SPLINE
SPL {X  -158.454, Y  +360.384, Z    +0.000, E1  +340.634, E3 -429443.801}
SPL {X  -159.737, Y  +373.507, Z    +0.000, E1  +349.689, E3 -429465.837}
SPL {X  -159.990, Y  +382.574, Z    +0.000, E1  +355.537, E3 -429472.525}
SPL {X  -159.990, Y  +389.909, Z    +0.000, E1  +360.662, E3 -429476.539}
SPL {X  -159.990, Y  +396.289, Z    +0.000, E1  +365.500, E3 -429480.319}
SPL {X  -159.990, Y  +407.941, Z    +0.000, E1  +374.126, E3 -429491.656}
SPL {X  -159.990, Y  +418.671, Z    +0.000, E1  +379.855, E3 -429511.072}
SPL {X  -159.990, Y  +429.878, Z    +0.000, E1  +383.330, E3 -429541.127}
SPL {X  -159.990, Y  +432.766, Z    +0.000, E1  +383.321, E3 -429555.350}
SPL {X  -159.990, Y  +434.794, Z    +0.000, E1  +383.304, E3 -429565.381}
SPL {X  -159.990, Y  +437.007, Z    +0.000, E1  +383.323, E3 -429576.234}
SPL {X  -159.990, Y  +439.778, Z    +0.000, E1  +383.323, E3 -429589.866}
SPL {X  -159.990, Y  +442.945, Z    +0.000, E1  +383.339, E3 -429605.430}
SPL {X  -159.990, Y  +446.037, Z    +0.000, E1  +383.324, E3 -429620.680}
SPL {X  -159.990, Y  +448.341, Z    +0.000, E1  +383.317, E3 -429631.998}
SPL {X  -159.990, Y  +450.345, Z    +0.000, E1  +383.316, E3 -429641.876}
SPL {X  -159.990, Y  +452.828, Z    +0.000, E1  +383.330, E3 -429654.075}
SPL {X  -159.990, Y  +456.338, Z    +0.000, E1  +383.359, E3 -429671.267}
SPL {X  -159.990, Y  +459.480, Z    +0.000, E1  +383.323, E3 -429686.809}
SPL {X  -159.990, Y  +461.803, Z    +0.000, E1  +383.322, E3 -429698.244}
SPL {X  -159.990, Y  +464.971, Z    +0.000, E1  +383.357, E3 -429713.750}
SPL {X  -159.990, Y  +467.934, Z    +0.000, E1  +383.321, E3 -429728.407}
SPL {X  -159.990, Y  +469.939, Z    +0.000, E1  +383.319, E3 -429738.269}
SPL {X  -159.990, Y  +472.144, Z    +0.000, E1  +383.327, E3 -429749.120}
SPL {X  -159.990, Y  +474.152, Z    +0.000, E1  +383.309, E3 -429759.072}
SPL {X  -159.990, Y  +475.762, Z    +0.000, E1  +383.308, E3 -429767.001}
SPL {X  -159.990, Y  +478.041, Z    +0.000, E1  +383.328, E3 -429778.177}
SPL {X  -159.990, Y  +480.905, Z    +0.000, E1  +383.327, E3 -429792.273}
SPL {X  -159.990, Y  +484.251, Z    +0.000, E1  +383.352, E3 -429808.688}
SPL {X  -159.990, Y  +488.031, Z    +0.000, E1  +383.345, E3 -429827.321}
SPL {X  -159.990, Y  +491.121, Z    +0.000, E1  +383.323, E3 -429842.567}
SPL {X  -159.990, Y  +493.610, Z    +0.000, E1  +383.323, E3 -429854.820}
SPL {X  -159.990, Y  +496.863, Z    +0.000, E1  +383.350, E3 -429870.780}
SPL {X  -159.990, Y  +499.995, Z    +0.000, E1  +383.324, E3 -429886.241}
SPL {X  -159.990, Y  +502.341, Z    +0.000, E1  +383.320, E3 -429897.800}
SPL {X  -159.990, Y  +505.377, Z    +0.000, E1  +383.346, E3 -429912.691}
SPL {X  -159.990, Y  +508.024, Z    +0.000, E1  +383.315, E3 -429925.773}
SPL {X  -159.990, Y  +510.344, Z    +0.000, E1  +383.327, E3 -429937.180}
SPL {X  -159.990, Y  +513.289, Z    +0.000, E1  +383.332, E3 -429951.670}
SPL {X  -159.990, Y  +516.195, Z    +0.000, E1  +383.325, E3 -429965.989}
SPL {X  -159.990, Y  +518.925, Z    +0.000, E1  +383.333, E3 -429979.352}
SPL {X  -159.990, Y  +521.408, Z    +0.000, E1  +383.329, E3 -429991.561}
SPL {X  -159.990, Y  +523.942, Z    +0.000, E1  +383.333, E3 -430004.054}
SPL {X  -159.990, Y  +526.221, Z    +0.000, E1  +383.314, E3 -430015.330}
SPL {X  -159.990, Y  +527.834, Z    +0.000, E1  +383.311, E3 -430023.280}
SPL {X  -159.990, Y  +529.993, Z    +0.000, E1  +383.329, E3 -430033.856}
SPL {X  -159.990, Y  +532.441, Z    +0.000, E1  +383.322, E3 -430045.907}
SPL {X  -159.990, Y  +534.618, Z    +0.000, E1  +383.322, E3 -430056.640}
SPL {X  -159.990, Y  +537.024, Z    +0.000, E1  +383.321, E3 -430068.502}
SPL {X  -159.990, Y  +539.129, Z    +0.000, E1  +383.310, E3 -430078.885}
SPL {X  -159.990, Y  +541.183, Z    +0.000, E1  +383.319, E3 -430088.982}
SPL {X  -159.990, Y  +543.647, Z    +0.000, E1  +383.325, E3 -430101.085}
SPL {X  -159.990, Y  +546.832, Z    +0.000, E1  +383.349, E3 -430116.708}
SPL {X  -159.990, Y  +549.756, Z    +0.000, E1  +383.320, E3 -430131.149}
SPL {X  -159.990, Y  +551.655, Z    +0.000, E1  +383.320, E3 -430140.499}
SPL {X  -159.990, Y  +553.711, Z    +0.000, E1  +383.317, E3 -430150.621}
SPL {X  -159.990, Y  +555.637, Z    +0.000, E1  +383.323, E3 -430160.090}
SPL {X  -159.990, Y  +558.758, Z    +0.000, E1  +383.351, E3 -430175.400}
SPL {X  -159.990, Y  +561.830, Z    +0.000, E1  +383.325, E3 -430190.573}
SPL {X  -159.990, Y  +564.273, Z    +0.000, E1  +383.325, E3 -430202.597}
SPL {X  -159.990, Y  +567.351, Z    +0.000, E1  +383.348, E3 -430217.693}
SPL {X  -159.990, Y  +570.314, Z    +0.000, E1  +383.326, E3 -430232.325}
SPL {X  -159.990, Y  +572.504, Z    +0.000, E1  +383.321, E3 -430243.110}
SPL {X  -159.990, Y  +575.653, Z    +0.000, E1  +383.355, E3 -430258.547}
SPL {X  -159.990, Y  +578.932, Z    +0.000, E1  +383.330, E3 -430274.730}
SPL {X  -159.990, Y  +581.497, Z    +0.000, E1  +383.329, E3 -430287.314}
SPL {X  -159.990, Y  +583.973, Z    +0.000, E1  +383.332, E3 -430299.499}
SPL {X  -159.990, Y  +586.877, Z    +0.000, E1  +383.349, E3 -430313.754}
SPL {X  -159.990, Y  +590.594, Z    +0.000, E1  +383.363, E3 -430332.004}
SPL {X  -159.990, Y  +593.847, Z    +0.000, E1  +383.340, E3 -430348.015}
SPL {X  -159.990, Y  +597.018, Z    +0.000, E1  +383.367, E3 -430363.546}
SPL {X  -159.990, Y  +599.887, Z    +0.000, E1  +383.341, E3 -430377.651}
SPL {X  -159.990, Y  +601.949, Z    +0.000, E1  +383.344, E3 -430387.777}
SPL {X  -159.990, Y  +605.106, Z    +0.000, E1  +383.383, E3 -430403.224}
SPL {X  -159.990, Y  +608.111, Z    +0.000, E1  +383.342, E3 -430418.075}
SPL {X  -159.990, Y  +610.073, Z    +0.000, E1  +383.343, E3 -430427.733}
SPL {X  -159.990, Y  +613.021, Z    +0.000, E1  +383.365, E3 -430442.203}
SPL {X  -159.990, Y  +615.657, Z    +0.000, E1  +383.331, E3 -430455.251}
SPL {X  -159.990, Y  +617.658, Z    +0.000, E1  +383.335, E3 -430465.093}
SPL {X  -159.990, Y  +620.788, Z    +0.000, E1  +383.368, E3 -430480.427}
SPL {X  -159.990, Y  +624.347, Z    +0.000, E1  +383.355, E3 -430497.947}
SPL {X  -159.990, Y  +627.144, Z    +0.000, E1  +383.340, E3 -430511.716}
SPL {X  -159.990, Y  +629.284, Z    +0.000, E1  +383.339, E3 -430522.224}
SPL {X  -159.990, Y  +631.206, Z    +0.000, E1  +383.337, E3 -430531.678}
SPL {X  -159.990, Y  +633.318, Z    +0.000, E1  +383.339, E3 -430542.082}
SPL {X  -159.990, Y  +635.650, Z    +0.000, E1  +383.339, E3 -430553.553}
SPL {X  -159.990, Y  +637.597, Z    +0.000, E1  +383.330, E3 -430563.176}
SPL {X  -159.990, Y  +640.369, Z    +0.000, E1  +383.354, E3 -430576.810}
SPL {X  -159.990, Y  +644.241, Z    +0.000, E1  +383.355, E3 -430595.922}
SPL {X  -159.990, Y  +648.287, Z    +0.000, E1  +383.349, E3 -430615.879}
SPL {X  -159.990, Y  +651.427, Z    +0.000, E1  +383.319, E3 -430631.374}
SPL {X  -159.990, Y  +653.536, Z    +0.000, E1  +383.313, E3 -430641.755}
SPL {X  -159.990, Y  +656.380, Z    +0.000, E1  +383.347, E3 -430655.691}
SPL {X  -159.990, Y  +659.180, Z    +0.000, E1  +383.314, E3 -430669.540}
SPL {X  -159.990, Y  +661.392, Z    +0.000, E1  +383.318, E3 -430680.433}
SPL {X  -159.990, Y  +663.662, Z    +0.000, E1  +383.322, E3 -430691.557}
SPL {X  -159.990, Y  +665.964, Z    +0.000, E1  +383.328, E3 -430702.848}
SPL {X  -159.990, Y  +668.989, Z    +0.000, E1  +383.359, E3 -430717.684}
SPL {X  -159.983, Y  +672.946, Z    +0.000, E1  +383.359, E3 -430737.165}
SPL {X  -159.924, Y  +676.110, Z    +0.000, E1  +383.320, E3 -430752.864}
SPL {X  -159.845, Y  +678.302, Z    +0.000, E1  +383.298, E3 -430763.766}
SPL {X  -159.760, Y  +680.081, Z    +0.000, E1  +383.288, E3 -430772.610}
SPL {X  -159.626, Y  +682.287, Z    +0.000, E1  +383.280, E3 -430783.581}
SPL {X  -159.462, Y  +684.486, Z    +0.000, E1  +383.258, E3 -430794.581}
SPL {X  -159.212, Y  +687.262, Z    +0.000, E1  +383.238, E3 -430808.485}
SPL {X  -158.971, Y  +689.529, Z    +0.000, E1  +383.181, E3 -430819.944}
SPL {X  -158.658, Y  +692.098, Z    +0.000, E1  +383.176, E3 -430832.851}
ENDSPLINE

SPLINE
SPL {X  -159.063, Y  +688.696, Z    +0.000, E1  +377.094, E3 -430875.070}
SPL {X  -159.987, Y  +672.488, Z    +0.000, E1  +365.638, E3 -430899.134}
SPL {X  -159.990, Y  +663.928, Z    +0.000, E1  +359.662, E3 -430904.929}
SPL {X  -159.990, Y  +658.009, Z    +0.000, E1  +355.226, E3 -430908.629}
SPL {X  -159.990, Y  +651.879, Z    +0.000, E1  +350.548, E3 -430913.691}
SPL {X  -159.990, Y  +637.832, Z    +0.000, E1  +341.694, E3 -430931.282}
SPL {X  -159.990, Y  +626.634, Z    +0.000, E1  +337.968, E3 -430962.136}
SPL {X  -159.990, Y  +624.622, Z    +0.000, E1  +337.980, E3 -430972.719}
SPL {X  -159.990, Y  +622.489, Z    +0.000, E1  +337.969, E3 -430983.886}
SPL {X  -159.990, Y  +619.955, Z    +0.000, E1  +337.968, E3 -430997.176}
SPL {X  -159.990, Y  +617.386, Z    +0.000, E1  +337.968, E3 -431010.650}
SPL {X  -159.990, Y  +614.863, Z    +0.000, E1  +337.969, E3 -431023.883}
SPL {X  -159.990, Y  +612.600, Z    +0.000, E1  +337.975, E3 -431035.767}
SPL {X  -159.990, Y  +610.646, Z    +0.000, E1  +337.979, E3 -431046.024}
SPL {X  -159.990, Y  +608.810, Z    +0.000, E1  +337.977, E3 -431055.657}
SPL {X  -159.990, Y  +605.804, Z    +0.000, E1  +337.936, E3 -431071.302}
SPL {X  -159.990, Y  +602.819, Z    +0.000, E1  +337.963, E3 -431086.974}
SPL {X  -159.990, Y  +600.642, Z    +0.000, E1  +337.968, E3 -431098.402}
SPL {X  -159.990, Y  +598.568, Z    +0.000, E1  +337.954, E3 -431109.194}
SPL {X  -159.990, Y  +595.493, Z    +0.000, E1  +337.930, E3 -431125.278}
SPL {X  -159.990, Y  +592.865, Z    +0.000, E1  +337.964, E3 -431139.106}
SPL {X  -159.990, Y  +590.803, Z    +0.000, E1  +337.954, E3 -431149.897}
SPL {X  -159.990, Y  +588.288, Z    +0.000, E1  +337.950, E3 -431163.061}
SPL {X  -159.990, Y  +586.040, Z    +0.000, E1  +337.954, E3 -431174.806}
SPL {X  -159.990, Y  +584.080, Z    +0.000, E1  +337.953, E3 -431185.066}
SPL {X  -159.990, Y  +581.924, Z    +0.000, E1  +337.949, E3 -431196.366}
SPL {X  -159.990, Y  +579.673, Z    +0.000, E1  +337.950, E3 -431208.165}
SPL {X  -159.990, Y  +576.961, Z    +0.000, E1  +337.936, E3 -431222.344}
SPL {X  -159.990, Y  +574.188, Z    +0.000, E1  +337.947, E3 -431236.891}
SPL {X  -159.990, Y  +571.954, Z    +0.000, E1  +337.959, E3 -431248.649}
SPL {X  -159.990, Y  +570.110, Z    +0.000, E1  +337.958, E3 -431258.299}
SPL {X  -159.990, Y  +568.165, Z    +0.000, E1  +337.957, E3 -431268.479}
SPL {X  -159.990, Y  +565.292, Z    +0.000, E1  +337.922, E3 -431283.457}
SPL {X  -159.990, Y  +562.598, Z    +0.000, E1  +337.958, E3 -431297.668}
SPL {X  -159.990, Y  +560.652, Z    +0.000, E1  +337.962, E3 -431307.880}
SPL {X  -159.990, Y  +558.143, Z    +0.000, E1  +337.928, E3 -431320.912}
SPL {X  -159.990, Y  +555.329, Z    +0.000, E1  +337.943, E3 -431335.656}
SPL {X  -159.990, Y  +553.115, Z    +0.000, E1  +337.946, E3 -431347.262}
SPL {X  -159.990, Y  +550.886, Z    +0.000, E1  +337.944, E3 -431358.943}
SPL {X  -159.990, Y  +548.568, Z    +0.000, E1  +337.944, E3 -431371.064}
SPL {X  -159.990, Y  +545.859, Z    +0.000, E1  +337.926, E3 -431385.213}
SPL {X  -159.990, Y  +542.390, Z    +0.000, E1  +337.914, E3 -431403.384}
SPL {X  -159.990, Y  +539.341, Z    +0.000, E1  +337.944, E3 -431419.406}
SPL {X  -159.990, Y  +536.935, Z    +0.000, E1  +337.942, E3 -431431.995}
SPL {X  -159.990, Y  +534.656, Z    +0.000, E1  +337.946, E3 -431443.939}
SPL {X  -159.990, Y  +532.453, Z    +0.000, E1  +337.944, E3 -431455.466}
SPL {X  -159.990, Y  +530.660, Z    +0.000, E1  +337.952, E3 -431464.869}
SPL {X  -159.990, Y  +528.702, Z    +0.000, E1  +337.939, E3 -431475.082}
SPL {X  -159.990, Y  +525.760, Z    +0.000, E1  +337.914, E3 -431490.423}
SPL {X  -159.990, Y  +522.838, Z    +0.000, E1  +337.933, E3 -431505.790}
SPL {X  -159.990, Y  +519.698, Z    +0.000, E1  +337.916, E3 -431522.173}
SPL {X  -159.990, Y  +517.251, Z    +0.000, E1  +337.946, E3 -431535.033}
SPL {X  -159.990, Y  +515.568, Z    +0.000, E1  +338.084, E3 -431545.130}
ENDSPLINE

SPLINE
SPL {X  -159.990, Y  +517.293, Z    +0.000, E1  +340.923, E3 -431561.428}
ENDSPLINE

SPLINE
SPL {X  -159.990, Y  +512.548, Z    +0.000, E1  +339.587, E3 -431577.003}
SPL {X  -159.990, Y  +508.660, Z    +0.000, E1  +338.515, E3 -431589.057}
SPL {X  -159.990, Y  +503.499, Z    +0.000, E1  +337.116, E3 -431604.136}
SPL {X  -159.990, Y  +498.406, Z    +0.000, E1  +335.789, E3 -431618.169}
SPL {X  -159.990, Y  +494.693, Z    +0.000, E1  +334.929, E3 -431628.637}
SPL {X  -159.990, Y  +491.649, Z    +0.000, E1  +334.596, E3 -431639.839}
SPL {X  -159.990, Y  +488.807, Z    +0.000, E1  +334.603, E3 -431652.564}
SPL {X  -159.990, Y  +486.070, Z    +0.000, E1  +334.601, E3 -431664.795}
SPL {X  -159.990, Y  +483.747, Z    +0.000, E1  +334.616, E3 -431675.207}
SPL {X  -159.990, Y  +481.038, Z    +0.000, E1  +334.588, E3 -431687.263}
SPL {X  -159.990, Y  +478.407, Z    +0.000, E1  +334.616, E3 -431699.077}
SPL {X  -159.990, Y  +475.940, Z    +0.000, E1  +334.597, E3 -431710.067}
SPL {X  -159.990, Y  +473.026, Z    +0.000, E1  +334.601, E3 -431723.097}
SPL {X  -159.990, Y  +470.047, Z    +0.000, E1  +334.598, E3 -431736.415}
SPL {X  -159.990, Y  +466.213, Z    +0.000, E1  +334.567, E3 -431753.495}
SPL {X  -159.990, Y  +462.520, Z    +0.000, E1  +334.600, E3 -431770.063}
SPL {X  -159.990, Y  +460.081, Z    +0.000, E1  +334.610, E3 -431780.965}
SPL {X  -159.990, Y  +457.497, Z    +0.000, E1  +334.597, E3 -431792.489}
SPL {X  -159.990, Y  +455.126, Z    +0.000, E1  +334.611, E3 -431803.098}
SPL {X  -159.990, Y  +453.438, Z    +0.000, E1  +334.615, E3 -431810.658}
SPL {X  -159.990, Y  +450.823, Z    +0.000, E1  +334.583, E3 -431822.277}
SPL {X  -159.990, Y  +446.894, Z    +0.000, E1  +334.572, E3 -431839.834}
SPL {X  -159.990, Y  +443.345, Z    +0.000, E1  +334.610, E3 -431855.842}
SPL {X  -159.990, Y  +441.077, Z    +0.000, E1  +334.631, E3 -431866.040}
SPL {X  -159.990, Y  +438.608, Z    +0.000, E1  +334.608, E3 -431877.037}
SPL {X  -159.990, Y  +434.852, Z    +0.000, E1  +334.585, E3 -431893.791}
SPL {X  -159.990, Y  +431.966, Z    +0.000, E1  +334.629, E3 -431906.789}
SPL {X  -159.990, Y  +429.079, Z    +0.000, E1  +334.593, E3 -431919.629}
SPL {X  -159.990, Y  +426.149, Z    +0.000, E1  +334.626, E3 -431932.791}
SPL {X  -159.990, Y  +423.417, Z    +0.000, E1  +334.600, E3 -431944.956}
SPL {X  -159.990, Y  +419.467, Z    +0.000, E1  +334.583, E3 -431962.591}
SPL {X  -159.990, Y  +416.355, Z    +0.000, E1  +334.625, E3 -431976.588}
SPL {X  -159.990, Y  +413.684, Z    +0.000, E1  +334.603, E3 -431988.495}
SPL {X  -159.990, Y  +410.645, Z    +0.000, E1  +334.615, E3 -432002.107}
SPL {X  -159.990, Y  +408.351, Z    +0.000, E1  +334.628, E3 -432012.393}
SPL {X  -159.990, Y  +406.574, Z    +0.000, E1  +334.625, E3 -432020.310}
SPL {X  -159.990, Y  +404.255, Z    +0.000, E1  +334.609, E3 -432030.646}
SPL {X  -159.990, Y  +401.103, Z    +0.000, E1  +334.596, E3 -432044.710}
SPL {X  -159.990, Y  +398.389, Z    +0.000, E1  +334.619, E3 -432056.906}
SPL {X  -159.990, Y  +395.411, Z    +0.000, E1  +334.600, E3 -432070.203}
SPL {X  -159.990, Y  +392.473, Z    +0.000, E1  +334.623, E3 -432083.388}
SPL {X  -159.990, Y  +390.187, Z    +0.000, E1  +334.622, E3 -432093.646}
SPL {X  -159.990, Y  +387.503, Z    +0.000, E1  +334.622, E3 -432105.641}
SPL {X  -159.990, Y  +384.711, Z    +0.000, E1  +334.612, E3 -432118.085}
SPL {X  -159.988, Y  +381.794, Z    +0.000, E1  +334.611, E3 -432131.120}
SPL {X  -159.958, Y  +379.279, Z    +0.000, E1  +334.625, E3 -432142.410}
SPL {X  -159.894, Y  +376.959, Z    +0.000, E1  +334.630, E3 -432152.854}
SPL {X  -159.765, Y  +374.027, Z    +0.000, E1  +334.633, E3 -432166.070}
SPL {X  -159.607, Y  +371.442, Z    +0.000, E1  +334.673, E3 -432177.845}
SPL {X  -159.379, Y  +368.534, Z    +0.000, E1  +334.684, E3 -432191.033}
SPL {X  -159.113, Y  +365.767, Z    +0.000, E1  +334.734, E3 -432203.672}
SPL {X  -158.798, Y  +363.007, Z    +0.000, E1  +334.761, E3 -432216.312}
SPL {X  -158.453, Y  +360.380, Z    +0.000, E1  +334.828, E3 -432228.457}
SPL {X  -158.127, Y  +358.155, Z    +0.000, E1  +334.874, E3 -432238.788}
SPL {X  -158.095, Y  +357.947, Z    +0.000, E1  +338.259, E3 -432270.360}
ENDSPLINE

SPLINE
SPL {X  -158.454, Y  +360.384, Z    +0.000, E1  +340.634, E3 -432282.511}
SPL {X  -159.737, Y  +373.507, Z    +0.000, E1  +349.689, E3 -432304.546}
SPL {X  -159.990, Y  +382.574, Z    +0.000, E1  +355.537, E3 -432311.234}
SPL {X  -159.990, Y  +387.496, Z    +0.000, E1  +358.996, E3 -432313.979}
SPL {X  -159.990, Y  +395.121, Z    +0.000, E1  +364.514, E3 -432318.292}
SPL {X  -159.990, Y  +407.941, Z    +0.000, E1  +374.126, E3 -432330.366}
SPL {X  -159.990, Y  +418.671, Z    +0.000, E1  +379.855, E3 -432349.782}
SPL {X  -159.990, Y  +429.878, Z    +0.000, E1  +383.330, E3 -432379.837}
SPL {X  -159.990, Y  +432.766, Z    +0.000, E1  +383.321, E3 -432394.060}
SPL {X  -159.990, Y  +434.794, Z    +0.000, E1  +383.304, E3 -432404.091}
SPL {X  -159.990, Y  +437.007, Z    +0.000, E1  +383.323, E3 -432414.943}
SPL {X  -159.990, Y  +439.778, Z    +0.000, E1  +383.323, E3 -432428.576}
SPL {X  -159.990, Y  +442.010, Z    +0.000, E1  +383.308, E3 -432439.597}
SPL {X  -159.990, Y  +443.729, Z    +0.000, E1  +383.310, E3 -432448.053}
SPL {X  -159.990, Y  +446.037, Z    +0.000, E1  +383.324, E3 -432459.390}
SPL {X  -159.990, Y  +448.341, Z    +0.000, E1  +383.317, E3 -432470.707}
SPL {X  -159.990, Y  +450.345, Z    +0.000, E1  +383.316, E3 -432480.585}
SPL {X  -159.990, Y  +452.828, Z    +0.000, E1  +383.330, E3 -432492.785}
SPL {X  -159.990, Y  +456.338, Z    +0.000, E1  +383.359, E3 -432509.977}
SPL {X  -159.990, Y  +459.480, Z    +0.000, E1  +383.323, E3 -432525.518}
SPL {X  -159.990, Y  +461.803, Z    +0.000, E1  +383.322, E3 -432536.954}
SPL {X  -159.990, Y  +464.971, Z    +0.000, E1  +383.357, E3 -432552.459}
SPL {X  -159.990, Y  +467.934, Z    +0.000, E1  +383.321, E3 -432567.117}
SPL {X  -159.990, Y  +469.939, Z    +0.000, E1  +383.319, E3 -432576.978}
SPL {X  -159.990, Y  +472.144, Z    +0.000, E1  +383.327, E3 -432587.829}
SPL {X  -159.990, Y  +474.152, Z    +0.000, E1  +383.309, E3 -432597.781}
SPL {X  -159.990, Y  +476.560, Z    +0.000, E1  +383.332, E3 -432609.589}
SPL {X  -159.990, Y  +478.770, Z    +0.000, E1  +383.306, E3 -432620.515}
SPL {X  -159.990, Y  +480.905, Z    +0.000, E1  +383.327, E3 -432630.983}
SPL {X  -159.990, Y  +484.251, Z    +0.000, E1  +383.352, E3 -432647.398}
SPL {X  -159.990, Y  +488.031, Z    +0.000, E1  +383.345, E3 -432666.031}
SPL {X  -159.990, Y  +491.121, Z    +0.000, E1  +383.323, E3 -432681.277}
SPL {X  -159.990, Y  +493.610, Z    +0.000, E1  +383.323, E3 -432693.530}
SPL {X  -159.990, Y  +496.863, Z    +0.000, E1  +383.350, E3 -432709.489}
SPL {X  -159.990, Y  +499.995, Z    +0.000, E1  +383.324, E3 -432724.951}
SPL {X  -159.990, Y  +502.341, Z    +0.000, E1  +383.320, E3 -432736.510}
SPL {X  -159.990, Y  +504.419, Z    +0.000, E1  +383.313, E3 -432746.752}
SPL {X  -159.990, Y  +507.187, Z    +0.000, E1  +383.346, E3 -432760.304}
SPL {X  -159.990, Y  +510.344, Z    +0.000, E1  +383.327, E3 -432775.890}
SPL {X  -159.990, Y  +512.484, Z    +0.000, E1  +383.309, E3 -432786.462}
SPL {X  -159.990, Y  +514.016, Z    +0.000, E1  +383.308, E3 -432794.011}
SPL {X  -159.990, Y  +516.195, Z    +0.000, E1  +383.325, E3 -432804.699}
SPL {X  -159.990, Y  +518.925, Z    +0.000, E1  +383.333, E3 -432818.062}
SPL {X  -159.990, Y  +521.408, Z    +0.000, E1  +383.329, E3 -432830.271}
SPL {X  -159.990, Y  +523.942, Z    +0.000, E1  +383.333, E3 -432842.764}
SPL {X  -159.990, Y  +527.007, Z    +0.000, E1  +383.339, E3 -432857.863}
SPL {X  -159.990, Y  +529.993, Z    +0.000, E1  +383.329, E3 -432872.566}
SPL {X  -159.990, Y  +532.441, Z    +0.000, E1  +383.322, E3 -432884.616}
SPL {X  -159.990, Y  +534.618, Z    +0.000, E1  +383.322, E3 -432895.349}
SPL {X  -159.990, Y  +537.024, Z    +0.000, E1  +383.321, E3 -432907.212}
SPL {X  -159.990, Y  +539.129, Z    +0.000, E1  +383.310, E3 -432917.595}
SPL {X  -159.990, Y  +541.183, Z    +0.000, E1  +383.319, E3 -432927.692}
SPL {X  -159.990, Y  +543.647, Z    +0.000, E1  +383.325, E3 -432939.795}
SPL {X  -159.990, Y  +546.832, Z    +0.000, E1  +383.349, E3 -432955.417}
SPL {X  -159.990, Y  +549.756, Z    +0.000, E1  +383.320, E3 -432969.858}
SPL {X  -159.990, Y  +551.655, Z    +0.000, E1  +383.320, E3 -432979.209}
SPL {X  -159.990, Y  +553.711, Z    +0.000, E1  +383.317, E3 -432989.331}
SPL {X  -159.990, Y  +555.637, Z    +0.000, E1  +383.323, E3 -432998.800}
SPL {X  -159.990, Y  +558.758, Z    +0.000, E1  +383.351, E3 -433014.109}
SPL {X  -159.990, Y  +561.830, Z    +0.000, E1  +383.325, E3 -433029.283}
SPL {X  -159.990, Y  +564.273, Z    +0.000, E1  +383.325, E3 -433041.307}
SPL {X  -159.990, Y  +567.351, Z    +0.000, E1  +383.348, E3 -433056.403}
SPL {X  -159.990, Y  +570.314, Z    +0.000, E1  +383.326, E3 -433071.035}
SPL {X  -159.990, Y  +572.504, Z    +0.000, E1  +383.321, E3 -433081.820}
SPL {X  -159.990, Y  +575.653, Z    +0.000, E1  +383.355, E3 -433097.257}
SPL {X  -159.990, Y  +578.932, Z    +0.000, E1  +383.330, E3 -433113.439}
SPL {X  -159.990, Y  +581.497, Z    +0.000, E1  +383.329, E3 -433126.024}
SPL {X  -159.990, Y  +583.973, Z    +0.000, E1  +383.332, E3 -433138.209}
SPL {X  -159.990, Y  +586.020, Z    +0.000, E1  +383.323, E3 -433148.293}
SPL {X  -159.990, Y  +587.711, Z    +0.000, E1  +383.318, E3 -433156.633}
SPL {X  -159.990, Y  +589.763, Z    +0.000, E1  +383.328, E3 -433166.709}
SPL {X  -159.990, Y  +591.698, Z    +0.000, E1  +383.324, E3 -433176.194}
SPL {X  -159.990, Y  +593.847, Z    +0.000, E1  +383.340, E3 -433186.724}
SPL {X  -159.990, Y  +597.018, Z    +0.000, E1  +383.367, E3 -433202.256}
SPL {X  -159.990, Y  +599.887, Z    +0.000, E1  +383.341, E3 -433216.360}
SPL {X  -159.990, Y  +601.949, Z    +0.000, E1  +383.344, E3 -433226.487}
SPL {X  -159.990, Y  +605.106, Z    +0.000, E1  +383.383, E3 -433241.933}
SPL {X  -159.990, Y  +608.111, Z    +0.000, E1  +383.342, E3 -433256.784}
SPL {X  -159.990, Y  +610.073, Z    +0.000, E1  +383.343, E3 -433266.442}
SPL {X  -159.990, Y  +613.021, Z    +0.000, E1  +383.365, E3 -433280.913}
SPL {X  -159.990, Y  +615.657, Z    +0.000, E1  +383.331, E3 -433293.961}
SPL {X  -159.990, Y  +617.658, Z    +0.000, E1  +383.335, E3 -433303.803}
SPL {X  -159.990, Y  +620.788, Z    +0.000, E1  +383.368, E3 -433319.136}
SPL {X  -159.990, Y  +624.347, Z    +0.000, E1  +383.355, E3 -433336.657}
SPL {X  -159.990, Y  +627.144, Z    +0.000, E1  +383.340, E3 -433350.426}
SPL {X  -159.990, Y  +629.284, Z    +0.000, E1  +383.339, E3 -433360.934}
SPL {X  -159.990, Y  +631.206, Z    +0.000, E1  +383.337, E3 -433370.387}
SPL {X  -159.990, Y  +633.318, Z    +0.000, E1  +383.339, E3 -433380.792}
SPL {X  -159.990, Y  +635.650, Z    +0.000, E1  +383.339, E3 -433392.263}
SPL {X  -159.990, Y  +637.597, Z    +0.000, E1  +383.330, E3 -433401.885}
SPL {X  -159.990, Y  +640.369, Z    +0.000, E1  +383.354, E3 -433415.520}
SPL {X  -159.990, Y  +644.241, Z    +0.000, E1  +383.355, E3 -433434.632}
SPL {X  -159.990, Y  +648.287, Z    +0.000, E1  +383.349, E3 -433454.589}
SPL {X  -159.990, Y  +651.427, Z    +0.000, E1  +383.319, E3 -433470.084}
SPL {X  -159.990, Y  +653.536, Z    +0.000, E1  +383.313, E3 -433480.465}
SPL {X  -159.990, Y  +656.380, Z    +0.000, E1  +383.347, E3 -433494.401}
SPL {X  -159.990, Y  +659.180, Z    +0.000, E1  +383.314, E3 -433508.249}
SPL {X  -159.990, Y  +661.392, Z    +0.000, E1  +383.318, E3 -433519.143}
SPL {X  -159.990, Y  +663.662, Z    +0.000, E1  +383.322, E3 -433530.267}
SPL {X  -159.990, Y  +665.964, Z    +0.000, E1  +383.328, E3 -433541.557}
SPL {X  -159.990, Y  +668.989, Z    +0.000, E1  +383.359, E3 -433556.393}
SPL {X  -159.983, Y  +672.946, Z    +0.000, E1  +383.359, E3 -433575.874}
SPL {X  -159.924, Y  +676.110, Z    +0.000, E1  +383.320, E3 -433591.574}
SPL {X  -159.801, Y  +679.265, Z    +0.000, E1  +383.327, E3 -433607.192}
SPL {X  -159.626, Y  +682.287, Z    +0.000, E1  +383.280, E3 -433622.291}
SPL {X  -159.462, Y  +684.486, Z    +0.000, E1  +383.258, E3 -433633.290}
SPL {X  -159.212, Y  +687.262, Z    +0.000, E1  +383.238, E3 -433647.194}
SPL {X  -158.971, Y  +689.529, Z    +0.000, E1  +383.181, E3 -433658.654}
SPL {X  -158.658, Y  +692.098, Z    +0.000, E1  +383.176, E3 -433671.561}
ENDSPLINE

SPLINE
SPL {X  -159.063, Y  +688.696, Z    +0.000, E1  +377.094, E3 -433713.779}
SPL {X  -159.987, Y  +672.488, Z    +0.000, E1  +365.638, E3 -433737.844}
SPL {X  -159.990, Y  +663.928, Z    +0.000, E1  +359.662, E3 -433743.639}
SPL {X  -159.990, Y  +658.009, Z    +0.000, E1  +355.226, E3 -433747.338}
SPL {X  -159.990, Y  +651.879, Z    +0.000, E1  +350.548, E3 -433752.401}
SPL {X  -159.990, Y  +637.832, Z    +0.000, E1  +341.694, E3 -433769.992}
SPL {X  -159.990, Y  +626.634, Z    +0.000, E1  +337.968, E3 -433800.845}
SPL {X  -159.990, Y  +624.622, Z    +0.000, E1  +337.980, E3 -433811.429}
SPL {X  -159.990, Y  +622.489, Z    +0.000, E1  +337.969, E3 -433822.595}
SPL {X  -159.990, Y  +619.267, Z    +0.000, E1  +337.938, E3 -433839.429}
SPL {X  -159.990, Y  +615.467, Z    +0.000, E1  +337.940, E3 -433859.366}
SPL {X  -159.990, Y  +612.600, Z    +0.000, E1  +337.975, E3 -433874.476}
SPL {X  -159.990, Y  +610.646, Z    +0.000, E1  +337.979, E3 -433884.734}
SPL {X  -159.990, Y  +608.810, Z    +0.000, E1  +337.977, E3 -433894.367}
SPL {X  -159.990, Y  +605.804, Z    +0.000, E1  +337.936, E3 -433910.012}
SPL {X  -159.990, Y  +602.819, Z    +0.000, E1  +337.963, E3 -433925.683}
SPL {X  -159.990, Y  +600.642, Z    +0.000, E1  +337.968, E3 -433937.111}
SPL {X  -159.990, Y  +598.568, Z    +0.000, E1  +337.954, E3 -433947.904}
SPL {X  -159.990, Y  +596.440, Z    +0.000, E1  +337.964, E3 -433959.086}
SPL {X  -159.990, Y  +593.768, Z    +0.000, E1  +337.929, E3 -433973.018}
SPL {X  -159.990, Y  +590.068, Z    +0.000, E1  +337.924, E3 -433992.387}
SPL {X  -159.990, Y  +586.620, Z    +0.000, E1  +337.935, E3 -434010.449}
SPL {X  -159.990, Y  +584.080, Z    +0.000, E1  +337.953, E3 -434023.776}
SPL {X  -159.990, Y  +581.924, Z    +0.000, E1  +337.949, E3 -434035.076}
SPL {X  -159.990, Y  +578.886, Z    +0.000, E1  +337.918, E3 -434050.930}
SPL {X  -159.990, Y  +576.252, Z    +0.000, E1  +337.962, E3 -434064.828}
SPL {X  -159.990, Y  +574.188, Z    +0.000, E1  +337.947, E3 -434075.601}
SPL {X  -159.990, Y  +571.954, Z    +0.000, E1  +337.959, E3 -434087.358}
SPL {X  -159.990, Y  +570.110, Z    +0.000, E1  +337.958, E3 -434097.009}
SPL {X  -159.990, Y  +568.165, Z    +0.000, E1  +337.957, E3 -434107.189}
SPL {X  -159.990, Y  +566.106, Z    +0.000, E1  +337.954, E3 -434117.972}
SPL {X  -159.990, Y  +563.259, Z    +0.000, E1  +337.929, E3 -434132.854}
SPL {X  -159.990, Y  +559.661, Z    +0.000, E1  +337.922, E3 -434151.677}
SPL {X  -159.990, Y  +555.965, Z    +0.000, E1  +337.915, E3 -434170.985}
SPL {X  -159.990, Y  +553.115, Z    +0.000, E1  +337.946, E3 -434185.971}
SPL {X  -159.990, Y  +550.886, Z    +0.000, E1  +337.944, E3 -434197.653}
SPL {X  -159.990, Y  +548.568, Z    +0.000, E1  +337.944, E3 -434209.774}
SPL {X  -159.990, Y  +546.537, Z    +0.000, E1  +337.948, E3 -434220.409}
SPL {X  -159.990, Y  +545.062, Z    +0.000, E1  +337.955, E3 -434228.167}
SPL {X  -159.990, Y  +543.060, Z    +0.000, E1  +337.943, E3 -434238.647}
SPL {X  -159.990, Y  +539.928, Z    +0.000, E1  +337.917, E3 -434254.988}
SPL {X  -159.990, Y  +536.935, Z    +0.000, E1  +337.942, E3 -434270.705}
SPL {X  -159.990, Y  +534.656, Z    +0.000, E1  +337.946, E3 -434282.649}
SPL {X  -159.990, Y  +532.453, Z    +0.000, E1  +337.944, E3 -434294.176}
SPL {X  -159.990, Y  +530.660, Z    +0.000, E1  +337.952, E3 -434303.578}
SPL {X  -159.990, Y  +528.702, Z    +0.000, E1  +337.939, E3 -434313.791}
SPL {X  -159.990, Y  +525.760, Z    +0.000, E1  +337.914, E3 -434329.133}
SPL {X  -159.990, Y  +522.838, Z    +0.000, E1  +337.933, E3 -434344.499}
SPL {X  -159.990, Y  +520.708, Z    +0.000, E1  +337.953, E3 -434355.693}
SPL {X  -159.990, Y  +518.216, Z    +0.000, E1  +337.909, E3 -434368.610}
SPL {X  -159.990, Y  +515.568, Z    +0.000, E1  +338.084, E3 -434383.839}
ENDSPLINE

SPLINE
SPL {X  -159.990, Y  +518.374, Z    +0.000, E1  +341.240, E3 -434396.427}
ENDSPLINE

SPLINE
SPL {X  -159.990, Y  +513.606, Z    +0.000, E1  +339.879, E3 -434412.338}
SPL {X  -159.990, Y  +508.660, Z    +0.000, E1  +338.515, E3 -434427.767}
SPL {X  -159.990, Y  +505.237, Z    +0.000, E1  +337.606, E3 -434438.024}
SPL {X  -159.990, Y  +501.963, Z    +0.000, E1  +336.712, E3 -434447.128}
SPL {X  -159.990, Y  +498.406, Z    +0.000, E1  +335.789, E3 -434456.879}
SPL {X  -159.990, Y  +494.693, Z    +0.000, E1  +334.929, E3 -434467.346}
SPL {X  -159.990, Y  +491.649, Z    +0.000, E1  +334.596, E3 -434478.549}
SPL {X  -159.990, Y  +488.807, Z    +0.000, E1  +334.603, E3 -434491.273}
SPL {X  -159.990, Y  +486.070, Z    +0.000, E1  +334.601, E3 -434503.504}
SPL {X  -159.990, Y  +483.747, Z    +0.000, E1  +334.616, E3 -434513.917}
SPL {X  -159.990, Y  +481.980, Z    +0.000, E1  +334.616, E3 -434521.815}
SPL {X  -159.990, Y  +479.252, Z    +0.000, E1  +334.588, E3 -434533.956}
SPL {X  -159.990, Y  +475.940, Z    +0.000, E1  +334.597, E3 -434548.777}
SPL {X  -159.990, Y  +473.026, Z    +0.000, E1  +334.601, E3 -434561.806}
SPL {X  -159.990, Y  +470.047, Z    +0.000, E1  +334.598, E3 -434575.125}
SPL {X  -159.990, Y  +466.213, Z    +0.000, E1  +334.567, E3 -434592.205}
SPL {X  -159.990, Y  +462.520, Z    +0.000, E1  +334.600, E3 -434608.773}
SPL {X  -159.990, Y  +460.081, Z    +0.000, E1  +334.610, E3 -434619.675}
SPL {X  -159.990, Y  +457.497, Z    +0.000, E1  +334.597, E3 -434631.199}
SPL {X  -159.990, Y  +455.126, Z    +0.000, E1  +334.611, E3 -434641.807}
SPL {X  -159.990, Y  +452.123, Z    +0.000, E1  +334.574, E3 -434655.165}
SPL {X  -159.990, Y  +448.503, Z    +0.000, E1  +334.590, E3 -434671.367}
SPL {X  -159.990, Y  +445.882, Z    +0.000, E1  +334.615, E3 -434683.169}
SPL {X  -159.990, Y  +443.345, Z    +0.000, E1  +334.610, E3 -434694.551}
SPL {X  -159.990, Y  +441.077, Z    +0.000, E1  +334.631, E3 -434704.750}
SPL {X  -159.990, Y  +438.608, Z    +0.000, E1  +334.608, E3 -434715.746}
SPL {X  -159.990, Y  +434.852, Z    +0.000, E1  +334.585, E3 -434732.501}
SPL {X  -159.990, Y  +430.645, Z    +0.000, E1  +334.586, E3 -434751.320}
SPL {X  -159.990, Y  +426.865, Z    +0.000, E1  +334.602, E3 -434768.250}
SPL {X  -159.990, Y  +424.251, Z    +0.000, E1  +334.625, E3 -434779.987}
SPL {X  -159.990, Y  +421.010, Z    +0.000, E1  +334.582, E3 -434794.402}
SPL {X  -159.990, Y  +417.103, Z    +0.000, E1  +334.600, E3 -434811.905}
SPL {X  -159.990, Y  +413.684, Z    +0.000, E1  +334.603, E3 -434827.205}
SPL {X  -159.990, Y  +410.645, Z    +0.000, E1  +334.615, E3 -434840.817}
SPL {X  -159.990, Y  +407.450, Z    +0.000, E1  +334.599, E3 -434855.065}
SPL {X  -159.990, Y  +403.513, Z    +0.000, E1  +334.580, E3 -434872.618}
SPL {X  -159.990, Y  +399.294, Z    +0.000, E1  +334.582, E3 -434891.498}
SPL {X  -159.990, Y  +395.411, Z    +0.000, E1  +334.600, E3 -434908.913}
SPL {X  -159.990, Y  +392.473, Z    +0.000, E1  +334.623, E3 -434922.098}
SPL {X  -159.990, Y  +390.187, Z    +0.000, E1  +334.622, E3 -434932.356}
SPL {X  -159.990, Y  +387.503, Z    +0.000, E1  +334.622, E3 -434944.351}
SPL {X  -159.990, Y  +384.711, Z    +0.000, E1  +334.612, E3 -434956.795}
SPL {X  -159.988, Y  +381.794, Z    +0.000, E1  +334.611, E3 -434969.829}
SPL {X  -159.958, Y  +379.279, Z    +0.000, E1  +334.625, E3 -434981.120}
SPL {X  -159.894, Y  +376.959, Z    +0.000, E1  +334.630, E3 -434991.564}
SPL {X  -159.765, Y  +374.027, Z    +0.000, E1  +334.633, E3 -435004.780}
SPL {X  -159.607, Y  +371.442, Z    +0.000, E1  +334.673, E3 -435016.555}
SPL {X  -159.379, Y  +368.534, Z    +0.000, E1  +334.684, E3 -435029.742}
SPL {X  -159.113, Y  +365.767, Z    +0.000, E1  +334.734, E3 -435042.382}
SPL {X  -158.869, Y  +363.595, Z    +0.000, E1  +334.770, E3 -435052.353}
SPL {X  -158.527, Y  +360.915, Z    +0.000, E1  +334.798, E3 -435064.659}
SPL {X  -158.127, Y  +358.155, Z    +0.000, E1  +334.874, E3 -435077.497}
SPL {X  -158.095, Y  +357.947, Z    +0.000, E1  +338.259, E3 -435109.070}
ENDSPLINE

SPLINE
SPL {X  -158.454, Y  +360.384, Z    +0.000, E1  +340.634, E3 -435121.221}
SPL {X  -159.737, Y  +373.507, Z    +0.000, E1  +349.689, E3 -435143.256}
SPL {X  -159.990, Y  +382.574, Z    +0.000, E1  +355.537, E3 -435149.944}
SPL {X  -159.990, Y  +389.909, Z    +0.000, E1  +360.662, E3 -435153.958}
SPL {X  -159.990, Y  +396.289, Z    +0.000, E1  +365.500, E3 -435157.739}
SPL {X  -159.990, Y  +407.941, Z    +0.000, E1  +374.126, E3 -435169.075}
SPL {X  -159.990, Y  +418.671, Z    +0.000, E1  +379.855, E3 -435188.492}
SPL {X  -159.990, Y  +428.534, Z    +0.000, E1  +383.299, E3 -435212.012}
SPL {X  -159.990, Y  +430.313, Z    +0.000, E1  +383.313, E3 -435220.725}
SPL {X  -159.990, Y  +432.766, Z    +0.000, E1  +383.321, E3 -435232.769}
SPL {X  -159.990, Y  +434.794, Z    +0.000, E1  +383.304, E3 -435242.801}
SPL {X  -159.990, Y  +437.007, Z    +0.000, E1  +383.323, E3 -435253.653}
SPL {X  -159.990, Y  +439.778, Z    +0.000, E1  +383.323, E3 -435267.285}
SPL {X  -159.990, Y  +442.010, Z    +0.000, E1  +383.308, E3 -435278.306}
SPL {X  -159.990, Y  +443.729, Z    +0.000, E1  +383.310, E3 -435286.763}
SPL {X  -159.990, Y  +446.037, Z    +0.000, E1  +383.324, E3 -435298.100}
SPL {X  -159.990, Y  +448.341, Z    +0.000, E1  +383.317, E3 -435309.417}
SPL {X  -159.990, Y  +450.345, Z    +0.000, E1  +383.316, E3 -435319.295}
SPL {X  -159.990, Y  +452.828, Z    +0.000, E1  +383.330, E3 -435331.495}
SPL {X  -159.990, Y  +455.244, Z    +0.000, E1  +383.317, E3 -435343.395}
SPL {X  -159.990, Y  +457.167, Z    +0.000, E1  +383.324, E3 -435352.825}
SPL {X  -159.990, Y  +459.480, Z    +0.000, E1  +383.323, E3 -435364.228}
SPL {X  -159.990, Y  +462.520, Z    +0.000, E1  +383.350, E3 -435379.133}
SPL {X  -159.990, Y  +465.602, Z    +0.000, E1  +383.328, E3 -435394.332}
SPL {X  -159.990, Y  +467.934, Z    +0.000, E1  +383.321, E3 -435405.827}
SPL {X  -159.990, Y  +469.939, Z    +0.000, E1  +383.319, E3 -435415.688}
SPL {X  -159.990, Y  +472.144, Z    +0.000, E1  +383.327, E3 -435426.539}
SPL {X  -159.990, Y  +474.994, Z    +0.000, E1  +383.334, E3 -435440.587}
SPL {X  -159.990, Y  +477.323, Z    +0.000, E1  +383.307, E3 -435452.102}
SPL {X  -159.990, Y  +479.553, Z    +0.000, E1  +383.328, E3 -435463.038}
SPL {X  -159.990, Y  +482.799, Z    +0.000, E1  +383.343, E3 -435478.977}
SPL {X  -159.990, Y  +485.299, Z    +0.000, E1  +383.310, E3 -435491.362}
SPL {X  -159.990, Y  +488.031, Z    +0.000, E1  +383.345, E3 -435504.741}
SPL {X  -159.990, Y  +491.121, Z    +0.000, E1  +383.323, E3 -435519.986}
SPL {X  -159.990, Y  +493.610, Z    +0.000, E1  +383.323, E3 -435532.239}
SPL {X  -159.990, Y  +495.794, Z    +0.000, E1  +383.312, E3 -435543.013}
SPL {X  -159.990, Y  +497.668, Z    +0.000, E1  +383.317, E3 -435552.223}
SPL {X  -159.990, Y  +499.995, Z    +0.000, E1  +383.324, E3 -435563.661}
SPL {X  -159.990, Y  +502.341, Z    +0.000, E1  +383.320, E3 -435575.220}
SPL {X  -159.990, Y  +504.419, Z    +0.000, E1  +383.313, E3 -435585.461}
SPL {X  -159.990, Y  +507.187, Z    +0.000, E1  +383.346, E3 -435599.014}
SPL {X  -159.990, Y  +510.344, Z    +0.000, E1  +383.327, E3 -435614.599}
SPL {X  -159.990, Y  +512.484, Z    +0.000, E1  +383.309, E3 -435625.172}
SPL {X  -159.990, Y  +514.016, Z    +0.000, E1  +383.308, E3 -435632.720}
SPL {X  -159.990, Y  +516.195, Z    +0.000, E1  +383.325, E3 -435643.408}
SPL {X  -159.990, Y  +518.925, Z    +0.000, E1  +383.333, E3 -435656.772}
SPL {X  -159.990, Y  +521.408, Z    +0.000, E1  +383.329, E3 -435668.981}
SPL {X  -159.990, Y  +523.942, Z    +0.000, E1  +383.333, E3 -435681.473}
SPL {X  -159.990, Y  +526.221, Z    +0.000, E1  +383.314, E3 -435692.749}
SPL {X  -159.990, Y  +527.834, Z    +0.000, E1  +383.311, E3 -435700.699}
SPL {X  -159.990, Y  +529.993, Z    +0.000, E1  +383.329, E3 -435711.275}
SPL {X  -159.990, Y  +532.441, Z    +0.000, E1  +383.322, E3 -435723.326}
SPL {X  -159.990, Y  +534.618, Z    +0.000, E1  +383.322, E3 -435734.059}
SPL {X  -159.990, Y  +537.024, Z    +0.000, E1  +383.321, E3 -435745.922}
SPL {X  -159.990, Y  +539.129, Z    +0.000, E1  +383.310, E3 -435756.304}
SPL {X  -159.990, Y  +541.183, Z    +0.000, E1  +383.319, E3 -435766.401}
SPL {X  -159.990, Y  +543.647, Z    +0.000, E1  +383.325, E3 -435778.504}
SPL {X  -159.990, Y  +546.832, Z    +0.000, E1  +383.349, E3 -435794.127}
SPL {X  -159.990, Y  +549.756, Z    +0.000, E1  +383.320, E3 -435808.568}
SPL {X  -159.990, Y  +551.655, Z    +0.000, E1  +383.320, E3 -435817.919}
SPL {X  -159.990, Y  +553.711, Z    +0.000, E1  +383.317, E3 -435828.041}
SPL {X  -159.990, Y  +555.637, Z    +0.000, E1  +383.323, E3 -435837.510}
SPL {X  -159.990, Y  +558.758, Z    +0.000, E1  +383.351, E3 -435852.819}
SPL {X  -159.990, Y  +561.830, Z    +0.000, E1  +383.325, E3 -435867.992}
SPL {X  -159.990, Y  +564.273, Z    +0.000, E1  +383.325, E3 -435880.017}
SPL {X  -159.990, Y  +567.351, Z    +0.000, E1  +383.348, E3 -435895.112}
SPL {X  -159.990, Y  +570.314, Z    +0.000, E1  +383.326, E3 -435909.745}
SPL {X  -159.990, Y  +572.504, Z    +0.000, E1  +383.321, E3 -435920.529}
SPL {X  -159.990, Y  +575.653, Z    +0.000, E1  +383.355, E3 -435935.966}
SPL {X  -159.990, Y  +578.932, Z    +0.000, E1  +383.330, E3 -435952.149}
SPL {X  -159.990, Y  +581.497, Z    +0.000, E1  +383.329, E3 -435964.734}
SPL {X  -159.990, Y  +583.973, Z    +0.000, E1  +383.332, E3 -435976.919}
SPL {X  -159.990, Y  +586.020, Z    +0.000, E1  +383.323, E3 -435987.003}
SPL {X  -159.990, Y  +587.711, Z    +0.000, E1  +383.318, E3 -435995.342}
SPL {X  -159.990, Y  +589.763, Z    +0.000, E1  +383.328, E3 -436005.419}
SPL {X  -159.990, Y  +591.698, Z    +0.000, E1  +383.324, E3 -436014.903}
SPL {X  -159.990, Y  +593.847, Z    +0.000, E1  +383.340, E3 -436025.434}
SPL {X  -159.990, Y  +597.018, Z    +0.000, E1  +383.367, E3 -436040.966}
SPL {X  -159.990, Y  +599.887, Z    +0.000, E1  +383.341, E3 -436055.070}
SPL {X  -159.990, Y  +601.949, Z    +0.000, E1  +383.344, E3 -436065.197}
SPL {X  -159.990, Y  +605.106, Z    +0.000, E1  +383.383, E3 -436080.643}
SPL {X  -159.990, Y  +608.111, Z    +0.000, E1  +383.342, E3 -436095.494}
SPL {X  -159.990, Y  +610.073, Z    +0.000, E1  +383.343, E3 -436105.152}
SPL {X  -159.990, Y  +612.330, Z    +0.000, E1  +383.340, E3 -436116.279}
SPL {X  -159.990, Y  +615.036, Z    +0.000, E1  +383.353, E3 -436129.567}
SPL {X  -159.990, Y  +618.481, Z    +0.000, E1  +383.366, E3 -436146.505}
SPL {X  -159.990, Y  +621.517, Z    +0.000, E1  +383.337, E3 -436161.488}
SPL {X  -159.990, Y  +623.764, Z    +0.000, E1  +383.335, E3 -436172.538}
SPL {X  -159.990, Y  +626.608, Z    +0.000, E1  +383.361, E3 -436186.463}
SPL {X  -159.990, Y  +629.284, Z    +0.000, E1  +383.339, E3 -436199.644}
SPL {X  -159.990, Y  +631.206, Z    +0.000, E1  +383.337, E3 -436209.097}
SPL {X  -159.990, Y  +633.318, Z    +0.000, E1  +383.339, E3 -436219.502}
SPL {X  -159.990, Y  +635.650, Z    +0.000, E1  +383.339, E3 -436230.972}
SPL {X  -159.990, Y  +637.597, Z    +0.000, E1  +383.330, E3 -436240.595}
SPL {X  -159.990, Y  +640.369, Z    +0.000, E1  +383.354, E3 -436254.229}
SPL {X  -159.990, Y  +644.241, Z    +0.000, E1  +383.355, E3 -436273.341}
SPL {X  -159.990, Y  +648.287, Z    +0.000, E1  +383.349, E3 -436293.298}
SPL {X  -159.990, Y  +651.427, Z    +0.000, E1  +383.319, E3 -436308.794}
SPL {X  -159.990, Y  +653.536, Z    +0.000, E1  +383.313, E3 -436319.175}
SPL {X  -159.990, Y  +656.380, Z    +0.000, E1  +383.347, E3 -436333.111}
SPL {X  -159.990, Y  +659.180, Z    +0.000, E1  +383.314, E3 -436346.959}
SPL {X  -159.990, Y  +661.392, Z    +0.000, E1  +383.318, E3 -436357.852}
SPL {X  -159.990, Y  +663.662, Z    +0.000, E1  +383.322, E3 -436368.977}
SPL {X  -159.990, Y  +665.964, Z    +0.000, E1  +383.328, E3 -436380.267}
SPL {X  -159.990, Y  +668.989, Z    +0.000, E1  +383.359, E3 -436395.103}
SPL {X  -159.983, Y  +672.946, Z    +0.000, E1  +383.359, E3 -436414.584}
SPL {X  -159.924, Y  +676.110, Z    +0.000, E1  +383.320, E3 -436430.283}
SPL {X  -159.845, Y  +678.302, Z    +0.000, E1  +383.298, E3 -436441.185}
SPL {X  -159.760, Y  +680.081, Z    +0.000, E1  +383.288, E3 -436450.029}
SPL {X  -159.626, Y  +682.287, Z    +0.000, E1  +383.280, E3 -436461.001}
SPL {X  -159.462, Y  +684.486, Z    +0.000, E1  +383.258, E3 -436472.000}
SPL {X  -159.289, Y  +686.457, Z    +0.000, E1  +383.223, E3 -436481.910}
SPL {X  -159.052, Y  +688.801, Z    +0.000, E1  +383.217, E3 -436493.645}
SPL {X  -158.658, Y  +692.098, Z    +0.000, E1  +383.176, E3 -436510.270}
ENDSPLINE

SPLINE
SPL {X  -158.898, Y  +690.164, Z    +0.000, E1  +378.236, E3 -436547.724}
SPL {X  -159.149, Y  +687.882, Z    +0.000, E1  +376.368, E3 -436555.012}
SPL {X  -159.987, Y  +672.488, Z    +0.000, E1  +365.638, E3 -436576.554}
SPL {X  -159.990, Y  +663.928, Z    +0.000, E1  +359.662, E3 -436582.348}
SPL {X  -159.990, Y  +658.009, Z    +0.000, E1  +355.226, E3 -436586.048}
SPL {X  -159.990, Y  +651.879, Z    +0.000, E1  +350.548, E3 -436591.111}
SPL {X  -159.990, Y  +637.832, Z    +0.000, E1  +341.694, E3 -436608.702}
SPL {X  -159.990, Y  +626.634, Z    +0.000, E1  +337.968, E3 -436639.555}
SPL {X  -159.990, Y  +624.622, Z    +0.000, E1  +337.980, E3 -436650.139}
SPL {X  -159.990, Y  +622.489, Z    +0.000, E1  +337.969, E3 -436661.305}
SPL {X  -159.990, Y  +619.267, Z    +0.000, E1  +337.938, E3 -436678.139}
SPL {X  -159.990, Y  +615.467, Z    +0.000, E1  +337.940, E3 -436698.076}
SPL {X  -159.990, Y  +612.600, Z    +0.000, E1  +337.975, E3 -436713.186}
SPL {X  -159.990, Y  +610.646, Z    +0.000, E1  +337.979, E3 -436723.443}
SPL {X  -159.990, Y  +608.810, Z    +0.000, E1  +337.977, E3 -436733.076}
SPL {X  -159.990, Y  +606.481, Z    +0.000, E1  +337.967, E3 -436745.252}
SPL {X  -159.990, Y  +603.419, Z    +0.000, E1  +337.936, E3 -436761.191}
SPL {X  -159.990, Y  +600.642, Z    +0.000, E1  +337.968, E3 -436775.821}
SPL {X  -159.990, Y  +598.568, Z    +0.000, E1  +337.954, E3 -436786.614}
SPL {X  -159.990, Y  +596.440, Z    +0.000, E1  +337.964, E3 -436797.795}
SPL {X  -159.990, Y  +593.768, Z    +0.000, E1  +337.929, E3 -436811.728}
SPL {X  -159.990, Y  +590.068, Z    +0.000, E1  +337.924, E3 -436831.097}
SPL {X  -159.990, Y  +586.620, Z    +0.000, E1  +337.935, E3 -436849.159}
SPL {X  -159.990, Y  +584.080, Z    +0.000, E1  +337.953, E3 -436862.485}
SPL {X  -159.990, Y  +581.924, Z    +0.000, E1  +337.949, E3 -436873.786}
SPL {X  -159.990, Y  +578.886, Z    +0.000, E1  +337.918, E3 -436889.640}
SPL {X  -159.990, Y  +576.252, Z    +0.000, E1  +337.962, E3 -436903.538}
SPL {X  -159.990, Y  +574.188, Z    +0.000, E1  +337.947, E3 -436914.311}
SPL {X  -159.990, Y  +571.954, Z    +0.000, E1  +337.959, E3 -436926.068}
SPL {X  -159.990, Y  +570.110, Z    +0.000, E1  +337.958, E3 -436935.719}
SPL {X  -159.990, Y  +568.165, Z    +0.000, E1  +337.957, E3 -436945.898}
SPL {X  -159.990, Y  +565.292, Z    +0.000, E1  +337.922, E3 -436960.876}
SPL {X  -159.990, Y  +562.598, Z    +0.000, E1  +337.958, E3 -436975.088}
SPL {X  -159.990, Y  +560.652, Z    +0.000, E1  +337.962, E3 -436985.300}
SPL {X  -159.990, Y  +558.143, Z    +0.000, E1  +337.928, E3 -436998.331}
SPL {X  -159.990, Y  +555.329, Z    +0.000, E1  +337.943, E3 -437013.076}
SPL {X  -159.990, Y  +553.115, Z    +0.000, E1  +337.946, E3 -437024.681}
SPL {X  -159.990, Y  +550.886, Z    +0.000, E1  +337.944, E3 -437036.362}
SPL {X  -159.990, Y  +548.568, Z    +0.000, E1  +337.944, E3 -437048.483}
SPL {X  -159.990, Y  +546.537, Z    +0.000, E1  +337.948, E3 -437059.118}
SPL {X  -159.990, Y  +545.062, Z    +0.000, E1  +337.955, E3 -437066.877}
SPL {X  -159.990, Y  +543.060, Z    +0.000, E1  +337.943, E3 -437077.356}
SPL {X  -159.990, Y  +539.928, Z    +0.000, E1  +337.917, E3 -437093.698}
SPL {X  -159.990, Y  +536.935, Z    +0.000, E1  +337.942, E3 -437109.415}
SPL {X  -159.990, Y  +534.656, Z    +0.000, E1  +337.946, E3 -437121.358}
SPL {X  -159.990, Y  +531.679, Z    +0.000, E1  +337.913, E3 -437136.872}
SPL {X  -159.990, Y  +527.941, Z    +0.000, E1  +337.907, E3 -437156.414}
SPL {X  -159.990, Y  +525.053, Z    +0.000, E1  +337.942, E3 -437171.605}
SPL {X  -159.990, Y  +522.838, Z    +0.000, E1  +337.933, E3 -437183.209}
SPL {X  -159.990, Y  +519.698, Z    +0.000, E1  +337.916, E3 -437199.592}
SPL {X  -159.990, Y  +517.251, Z    +0.000, E1  +337.946, E3 -437212.452}
SPL {X  -159.990, Y  +515.568, Z    +0.000, E1  +338.084, E3 -437222.549}
ENDSPLINE

SPLINE
SPL {X  -159.990, Y  +517.293, Z    +0.000, E1  +340.923, E3 -437238.847}
ENDSPLINE

SPLINE
SPL {X  -159.990, Y  +512.548, Z    +0.000, E1  +339.587, E3 -437254.422}
SPL {X  -159.990, Y  +508.660, Z    +0.000, E1  +338.515, E3 -437266.477}
SPL {X  -159.990, Y  +503.499, Z    +0.000, E1  +337.116, E3 -437281.556}
SPL {X  -159.990, Y  +498.406, Z    +0.000, E1  +335.789, E3 -437295.589}
SPL {X  -159.990, Y  +494.693, Z    +0.000, E1  +334.929, E3 -437306.056}
SPL {X  -159.990, Y  +491.649, Z    +0.000, E1  +334.596, E3 -437317.259}
SPL {X  -159.990, Y  +488.807, Z    +0.000, E1  +334.603, E3 -437329.983}
SPL {X  -159.990, Y  +486.070, Z    +0.000, E1  +334.601, E3 -437342.214}
SPL {X  -159.990, Y  +483.747, Z    +0.000, E1  +334.616, E3 -437352.627}
SPL {X  -159.990, Y  +481.038, Z    +0.000, E1  +334.588, E3 -437364.682}
SPL {X  -159.990, Y  +478.407, Z    +0.000, E1  +334.616, E3 -437376.496}
SPL {X  -159.990, Y  +475.940, Z    +0.000, E1  +334.597, E3 -437387.486}
SPL {X  -159.990, Y  +473.026, Z    +0.000, E1  +334.601, E3 -437400.516}
SPL {X  -159.990, Y  +470.047, Z    +0.000, E1  +334.598, E3 -437413.835}
SPL {X  -159.990, Y  +467.082, Z    +0.000, E1  +334.601, E3 -437427.082}
SPL {X  -159.990, Y  +464.919, Z    +0.000, E1  +334.619, E3 -437436.808}
SPL {X  -159.990, Y  +462.520, Z    +0.000, E1  +334.600, E3 -437447.483}
SPL {X  -159.990, Y  +460.081, Z    +0.000, E1  +334.610, E3 -437458.384}
SPL {X  -159.990, Y  +457.497, Z    +0.000, E1  +334.597, E3 -437469.909}
SPL {X  -159.990, Y  +454.323, Z    +0.000, E1  +334.588, E3 -437484.068}
SPL {X  -159.990, Y  +451.400, Z    +0.000, E1  +334.603, E3 -437497.159}
SPL {X  -159.990, Y  +448.503, Z    +0.000, E1  +334.590, E3 -437510.076}
SPL {X  -159.990, Y  +445.882, Z    +0.000, E1  +334.615, E3 -437521.879}
SPL {X  -159.990, Y  +443.345, Z    +0.000, E1  +334.610, E3 -437533.261}
SPL {X  -159.990, Y  +441.077, Z    +0.000, E1  +334.631, E3 -437543.459}
SPL {X  -159.990, Y  +438.608, Z    +0.000, E1  +334.608, E3 -437554.456}
SPL {X  -159.990, Y  +434.852, Z    +0.000, E1  +334.585, E3 -437571.211}
SPL {X  -159.990, Y  +430.645, Z    +0.000, E1  +334.586, E3 -437590.030}
SPL {X  -159.990, Y  +426.865, Z    +0.000, E1  +334.602, E3 -437606.960}
SPL {X  -159.990, Y  +424.251, Z    +0.000, E1  +334.625, E3 -437618.697}
SPL {X  -159.990, Y  +421.010, Z    +0.000, E1  +334.582, E3 -437633.112}
SPL {X  -159.990, Y  +417.103, Z    +0.000, E1  +334.600, E3 -437650.615}
SPL {X  -159.990, Y  +414.457, Z    +0.000, E1  +334.626, E3 -437662.503}
SPL {X  -159.990, Y  +411.297, Z    +0.000, E1  +334.587, E3 -437676.560}
SPL {X  -159.990, Y  +407.450, Z    +0.000, E1  +334.599, E3 -437693.775}
SPL {X  -159.990, Y  +404.255, Z    +0.000, E1  +334.609, E3 -437708.065}
SPL {X  -159.990, Y  +401.103, Z    +0.000, E1  +334.596, E3 -437722.130}
SPL {X  -159.990, Y  +397.743, Z    +0.000, E1  +334.600, E3 -437737.180}
SPL {X  -159.990, Y  +394.848, Z    +0.000, E1  +334.621, E3 -437750.181}
SPL {X  -159.990, Y  +392.473, Z    +0.000, E1  +334.623, E3 -437760.808}
SPL {X  -159.990, Y  +390.187, Z    +0.000, E1  +334.622, E3 -437771.066}
SPL {X  -159.990, Y  +387.503, Z    +0.000, E1  +334.622, E3 -437783.061}
SPL {X  -159.990, Y  +384.711, Z    +0.000, E1  +334.612, E3 -437795.504}
SPL {X  -159.988, Y  +381.794, Z    +0.000, E1  +334.611, E3 -437808.539}
SPL {X  -159.958, Y  +379.279, Z    +0.000, E1  +334.625, E3 -437819.829}
SPL {X  -159.894, Y  +376.959, Z    +0.000, E1  +334.630, E3 -437830.274}
SPL {X  -159.765, Y  +374.027, Z    +0.000, E1  +334.633, E3 -437843.489}
SPL {X  -159.607, Y  +371.442, Z    +0.000, E1  +334.673, E3 -437855.264}
SPL {X  -159.379, Y  +368.534, Z    +0.000, E1  +334.684, E3 -437868.452}
SPL {X  -159.113, Y  +365.767, Z    +0.000, E1  +334.734, E3 -437881.092}
SPL {X  -158.798, Y  +363.007, Z    +0.000, E1  +334.761, E3 -437893.732}
SPL {X  -158.453, Y  +360.380, Z    +0.000, E1  +334.828, E3 -437905.876}
SPL {X  -158.127, Y  +358.155, Z    +0.000, E1  +334.874, E3 -437916.207}
SPL {X  -158.095, Y  +357.947, Z    +0.000, E1  +338.259, E3 -437947.779}
ENDSPLINE

SPLINE
SPL {X  -158.454, Y  +360.384, Z    +0.000, E1  +340.634, E3 -437959.930}
SPL {X  -159.737, Y  +373.507, Z    +0.000, E1  +349.689, E3 -437981.966}
SPL {X  -159.990, Y  +382.574, Z    +0.000, E1  +355.537, E3 -437988.654}
SPL {X  -159.990, Y  +389.909, Z    +0.000, E1  +360.662, E3 -437992.668}
SPL {X  -159.990, Y  +396.289, Z    +0.000, E1  +365.500, E3 -437996.448}
SPL {X  -159.990, Y  +407.941, Z    +0.000, E1  +374.126, E3 -438007.785}
SPL {X  -159.990, Y  +418.671, Z    +0.000, E1  +379.855, E3 -438027.201}
SPL {X  -159.990, Y  +429.878, Z    +0.000, E1  +383.330, E3 -438057.256}
SPL {X  -159.990, Y  +432.766, Z    +0.000, E1  +383.321, E3 -438071.479}
SPL {X  -159.990, Y  +435.585, Z    +0.000, E1  +383.327, E3 -438085.359}
SPL {X  -159.990, Y  +439.169, Z    +0.000, E1  +383.353, E3 -438102.941}
SPL {X  -159.990, Y  +442.945, Z    +0.000, E1  +383.339, E3 -438121.559}
SPL {X  -159.990, Y  +446.037, Z    +0.000, E1  +383.324, E3 -438136.809}
SPL {X  -159.990, Y  +448.341, Z    +0.000, E1  +383.317, E3 -438148.127}
SPL {X  -159.990, Y  +450.968, Z    +0.000, E1  +383.336, E3 -438161.042}
SPL {X  -159.990, Y  +454.421, Z    +0.000, E1  +383.348, E3 -438177.992}
SPL {X  -159.990, Y  +457.167, Z    +0.000, E1  +383.324, E3 -438191.535}
SPL {X  -159.990, Y  +459.480, Z    +0.000, E1  +383.323, E3 -438202.938}
SPL {X  -159.990, Y  +462.520, Z    +0.000, E1  +383.350, E3 -438217.842}
SPL {X  -159.990, Y  +465.602, Z    +0.000, E1  +383.328, E3 -438233.042}
SPL {X  -159.990, Y  +467.934, Z    +0.000, E1  +383.321, E3 -438244.536}
SPL {X  -159.990, Y  +469.939, Z    +0.000, E1  +383.319, E3 -438254.398}
SPL {X  -159.990, Y  +472.144, Z    +0.000, E1  +383.327, E3 -438265.249}
SPL {X  -159.990, Y  +474.994, Z    +0.000, E1  +383.334, E3 -438279.297}
SPL {X  -159.990, Y  +477.323, Z    +0.000, E1  +383.307, E3 -438290.812}
SPL {X  -159.990, Y  +479.553, Z    +0.000, E1  +383.328, E3 -438301.747}
SPL {X  -159.990, Y  +482.799, Z    +0.000, E1  +383.343, E3 -438317.687}
SPL {X  -159.990, Y  +485.299, Z    +0.000, E1  +383.310, E3 -438330.072}
SPL {X  -159.990, Y  +487.362, Z    +0.000, E1  +383.320, E3 -438340.205}
SPL {X  -159.990, Y  +490.503, Z    +0.000, E1  +383.351, E3 -438355.601}
SPL {X  -159.990, Y  +493.610, Z    +0.000, E1  +383.323, E3 -438370.949}
SPL {X  -159.990, Y  +495.794, Z    +0.000, E1  +383.312, E3 -438381.722}
SPL {X  -159.990, Y  +497.668, Z    +0.000, E1  +383.317, E3 -438390.932}
SPL {X  -159.990, Y  +499.995, Z    +0.000, E1  +383.324, E3 -438402.370}
SPL {X  -159.990, Y  +502.341, Z    +0.000, E1  +383.320, E3 -438413.929}
SPL {X  -159.990, Y  +504.419, Z    +0.000, E1  +383.313, E3 -438424.171}
SPL {X  -159.990, Y  +507.187, Z    +0.000, E1  +383.346, E3 -438437.724}
SPL {X  -159.990, Y  +510.344, Z    +0.000, E1  +383.327, E3 -438453.309}
SPL {X  -159.990, Y  +512.484, Z    +0.000, E1  +383.309, E3 -438463.881}
SPL {X  -159.990, Y  +514.016, Z    +0.000, E1  +383.308, E3 -438471.430}
SPL {X  -159.990, Y  +516.195, Z    +0.000, E1  +383.325, E3 -438482.118}
SPL {X  -159.990, Y  +518.925, Z    +0.000, E1  +383.333, E3 -438495.481}
SPL {X  -159.990, Y  +521.408, Z    +0.000, E1  +383.329, E3 -438507.690}
SPL {X  -159.990, Y  +523.942, Z    +0.000, E1  +383.333, E3 -438520.183}
SPL {X  -159.990, Y  +527.007, Z    +0.000, E1  +383.339, E3 -438535.282}
SPL {X  -159.990, Y  +529.993, Z    +0.000, E1  +383.329, E3 -438549.985}
SPL {X  -159.990, Y  +532.441, Z    +0.000, E1  +383.322, E3 -438562.036}
SPL {X  -159.990, Y  +534.618, Z    +0.000, E1  +383.322, E3 -438572.769}
SPL {X  -159.990, Y  +537.024, Z    +0.000, E1  +383.321, E3 -438584.631}
SPL {X  -159.990, Y  +539.129, Z    +0.000, E1  +383.310, E3 -438595.014}
SPL {X  -159.990, Y  +541.183, Z    +0.000, E1  +383.319, E3 -438605.111}
SPL {X  -159.990, Y  +543.647, Z    +0.000, E1  +383.325, E3 -438617.214}
SPL {X  -159.990, Y  +545.957, Z    +0.000, E1  +383.318, E3 -438628.594}
SPL {X  -159.990, Y  +548.912, Z    +0.000, E1  +383.354, E3 -438643.053}
SPL {X  -159.990, Y  +551.655, Z    +0.000, E1  +383.320, E3 -438656.628}
SPL {X  -159.990, Y  +553.711, Z    +0.000, E1  +383.317, E3 -438666.750}
SPL {X  -159.990, Y  +556.481, Z    +0.000, E1  +383.354, E3 -438680.312}
SPL {X  -159.990, Y  +559.475, Z    +0.000, E1  +383.321, E3 -438695.118}
SPL {X  -159.990, Y  +561.830, Z    +0.000, E1  +383.325, E3 -438706.702}
SPL {X  -159.990, Y  +564.273, Z    +0.000, E1  +383.325, E3 -438718.726}
SPL {X  -159.990, Y  +566.342, Z    +0.000, E1  +383.314, E3 -438728.931}
SPL {X  -159.990, Y  +568.184, Z    +0.000, E1  +383.317, E3 -438737.992}
SPL {X  -159.990, Y  +570.314, Z    +0.000, E1  +383.326, E3 -438748.454}
SPL {X  -159.990, Y  +573.444, Z    +0.000, E1  +383.356, E3 -438763.794}
SPL {X  -159.990, Y  +576.445, Z    +0.000, E1  +383.320, E3 -438778.642}
SPL {X  -159.990, Y  +578.932, Z    +0.000, E1  +383.330, E3 -438790.859}
SPL {X  -159.990, Y  +581.497, Z    +0.000, E1  +383.329, E3 -438803.443}
SPL {X  -159.990, Y  +583.973, Z    +0.000, E1  +383.332, E3 -438815.628}
SPL {X  -159.990, Y  +586.877, Z    +0.000, E1  +383.349, E3 -438829.883}
SPL {X  -159.990, Y  +590.594, Z    +0.000, E1  +383.363, E3 -438848.133}
SPL {X  -159.990, Y  +593.847, Z    +0.000, E1  +383.340, E3 -438864.144}
SPL {X  -159.990, Y  +596.027, Z    +0.000, E1  +383.330, E3 -438874.890}
SPL {X  -159.990, Y  +599.017, Z    +0.000, E1  +383.373, E3 -438889.455}
SPL {X  -159.990, Y  +601.949, Z    +0.000, E1  +383.344, E3 -438903.906}
SPL {X  -159.990, Y  +604.315, Z    +0.000, E1  +383.350, E3 -438915.532}
SPL {X  -159.990, Y  +607.388, Z    +0.000, E1  +383.369, E3 -438930.596}
SPL {X  -159.990, Y  +610.073, Z    +0.000, E1  +383.343, E3 -438943.862}
SPL {X  -159.990, Y  +612.330, Z    +0.000, E1  +383.340, E3 -438954.989}
SPL {X  -159.990, Y  +615.036, Z    +0.000, E1  +383.353, E3 -438968.276}
SPL {X  -159.990, Y  +618.481, Z    +0.000, E1  +383.366, E3 -438985.214}
SPL {X  -159.990, Y  +621.517, Z    +0.000, E1  +383.337, E3 -439000.197}
SPL {X  -159.990, Y  +623.764, Z    +0.000, E1  +383.335, E3 -439011.248}
SPL {X  -159.990, Y  +626.608, Z    +0.000, E1  +383.361, E3 -439025.173}
SPL {X  -159.990, Y  +630.271, Z    +0.000, E1  +383.375, E3 -439043.134}
SPL {X  -159.990, Y  +633.318, Z    +0.000, E1  +383.339, E3 -439058.211}
SPL {X  -159.990, Y  +635.650, Z    +0.000, E1  +383.339, E3 -439069.682}
SPL {X  -159.990, Y  +638.406, Z    +0.000, E1  +383.354, E3 -439083.249}
SPL {X  -159.990, Y  +641.831, Z    +0.000, E1  +383.342, E3 -439100.196}
SPL {X  -159.990, Y  +644.884, Z    +0.000, E1  +383.324, E3 -439115.283}
SPL {X  -159.990, Y  +647.550, Z    +0.000, E1  +383.318, E3 -439128.450}
SPL {X  -159.990, Y  +650.790, Z    +0.000, E1  +383.346, E3 -439144.317}
SPL {X  -159.990, Y  +654.543, Z    +0.000, E1  +383.348, E3 -439162.770}
SPL {X  -159.990, Y  +658.319, Z    +0.000, E1  +383.349, E3 -439181.359}
SPL {X  -159.990, Y  +661.392, Z    +0.000, E1  +383.318, E3 -439196.562}
SPL {X  -159.990, Y  +663.662, Z    +0.000, E1  +383.322, E3 -439207.686}
SPL {X  -159.990, Y  +665.964, Z    +0.000, E1  +383.328, E3 -439218.977}
SPL {X  -159.990, Y  +667.870, Z    +0.000, E1  +383.320, E3 -439228.384}
SPL {X  -159.990, Y  +669.861, Z    +0.000, E1  +383.321, E3 -439238.185}
SPL {X  -159.990, Y  +671.893, Z    +0.000, E1  +383.319, E3 -439248.193}
SPL {X  -159.974, Y  +673.789, Z    +0.000, E1  +383.323, E3 -439257.508}
SPL {X  -159.924, Y  +676.110, Z    +0.000, E1  +383.320, E3 -439268.993}
SPL {X  -159.801, Y  +679.265, Z    +0.000, E1  +383.327, E3 -439284.612}
SPL {X  -159.626, Y  +682.287, Z    +0.000, E1  +383.280, E3 -439299.710}
SPL {X  -159.462, Y  +684.486, Z    +0.000, E1  +383.258, E3 -439310.710}
SPL {X  -159.289, Y  +686.457, Z    +0.000, E1  +383.223, E3 -439320.620}
SPL {X  -159.052, Y  +688.801, Z    +0.000, E1  +383.217, E3 -439332.355}
SPL {X  -158.658, Y  +692.098, Z    +0.000, E1  +383.176, E3 -439348.980}
ENDSPLINE

SPLINE
SPL {X  -159.063, Y  +688.696, Z    +0.000, E1  +377.094, E3 -439391.199}
SPL {X  -159.957, Y  +674.769, Z    +0.000, E1  +367.092, E3 -439413.580}
SPL {X  -159.990, Y  +671.516, Z    +0.000, E1  +364.944, E3 -439415.966}
SPL {X  -159.990, Y  +663.928, Z    +0.000, E1  +359.662, E3 -439421.058}
SPL {X  -159.990, Y  +658.009, Z    +0.000, E1  +355.226, E3 -439424.758}
SPL {X  -159.990, Y  +651.879, Z    +0.000, E1  +350.548, E3 -439429.820}
SPL {X  -159.990, Y  +637.832, Z    +0.000, E1  +341.694, E3 -439447.411}
SPL {X  -159.990, Y  +626.634, Z    +0.000, E1  +337.968, E3 -439478.265}
SPL {X  -159.990, Y  +624.622, Z    +0.000, E1  +337.980, E3 -439488.848}
SPL {X  -159.990, Y  +622.489, Z    +0.000, E1  +337.969, E3 -439500.015}
SPL {X  -159.990, Y  +619.955, Z    +0.000, E1  +337.968, E3 -439513.305}
SPL {X  -159.990, Y  +617.386, Z    +0.000, E1  +337.968, E3 -439526.779}
SPL {X  -159.990, Y  +614.863, Z    +0.000, E1  +337.969, E3 -439540.012}
SPL {X  -159.990, Y  +612.600, Z    +0.000, E1  +337.975, E3 -439551.896}
SPL {X  -159.990, Y  +610.646, Z    +0.000, E1  +337.979, E3 -439562.153}
SPL {X  -159.990, Y  +608.810, Z    +0.000, E1  +337.977, E3 -439571.786}
SPL {X  -159.990, Y  +605.804, Z    +0.000, E1  +337.936, E3 -439587.431}
SPL {X  -159.990, Y  +602.819, Z    +0.000, E1  +337.963, E3 -439603.103}
SPL {X  -159.990, Y  +600.642, Z    +0.000, E1  +337.968, E3 -439614.531}
SPL {X  -159.990, Y  +598.568, Z    +0.000, E1  +337.954, E3 -439625.323}
SPL {X  -159.990, Y  +596.440, Z    +0.000, E1  +337.964, E3 -439636.505}
SPL {X  -159.990, Y  +593.768, Z    +0.000, E1  +337.929, E3 -439650.438}
SPL {X  -159.990, Y  +590.068, Z    +0.000, E1  +337.924, E3 -439669.806}
SPL {X  -159.990, Y  +586.620, Z    +0.000, E1  +337.935, E3 -439687.869}
SPL {X  -159.990, Y  +584.080, Z    +0.000, E1  +337.953, E3 -439701.195}
SPL {X  -159.990, Y  +581.924, Z    +0.000, E1  +337.949, E3 -439712.495}
SPL {X  -159.990, Y  +578.886, Z    +0.000, E1  +337.918, E3 -439728.349}
SPL {X  -159.990, Y  +576.252, Z    +0.000, E1  +337.962, E3 -439742.247}
SPL {X  -159.990, Y  +574.188, Z    +0.000, E1  +337.947, E3 -439753.020}
SPL {X  -159.990, Y  +571.954, Z    +0.000, E1  +337.959, E3 -439764.778}
SPL {X  -159.990, Y  +570.110, Z    +0.000, E1  +337.958, E3 -439774.428}
SPL {X  -159.990, Y  +568.165, Z    +0.000, E1  +337.957, E3 -439784.608}
SPL {X  -159.990, Y  +566.106, Z    +0.000, E1  +337.954, E3 -439795.391}
SPL {X  -159.990, Y  +563.259, Z    +0.000, E1  +337.929, E3 -439810.273}
SPL {X  -159.990, Y  +559.661, Z    +0.000, E1  +337.922, E3 -439829.096}
SPL {X  -159.990, Y  +555.965, Z    +0.000, E1  +337.915, E3 -439848.405}
SPL {X  -159.990, Y  +553.115, Z    +0.000, E1  +337.946, E3 -439863.391}
SPL {X  -159.990, Y  +550.886, Z    +0.000, E1  +337.944, E3 -439875.072}
SPL {X  -159.990, Y  +548.568, Z    +0.000, E1  +337.944, E3 -439887.193}
SPL {X  -159.990, Y  +546.537, Z    +0.000, E1  +337.948, E3 -439897.828}
SPL {X  -159.990, Y  +545.062, Z    +0.000, E1  +337.955, E3 -439905.587}
SPL {X  -159.990, Y  +543.060, Z    +0.000, E1  +337.943, E3 -439916.066}
SPL {X  -159.990, Y  +539.928, Z    +0.000, E1  +337.917, E3 -439932.407}
SPL {X  -159.990, Y  +536.935, Z    +0.000, E1  +337.942, E3 -439948.124}
SPL {X  -159.990, Y  +534.656, Z    +0.000, E1  +337.946, E3 -439960.068}
SPL {X  -159.990, Y  +531.679, Z    +0.000, E1  +337.913, E3 -439975.582}
SPL {X  -159.990, Y  +527.941, Z    +0.000, E1  +337.907, E3 -439995.124}
SPL {X  -159.990, Y  +524.425, Z    +0.000, E1  +337.922, E3 -440013.580}
SPL {X  -159.990, Y  +521.385, Z    +0.000, E1  +337.932, E3 -440029.522}
SPL {X  -159.990, Y  +518.216, Z    +0.000, E1  +337.909, E3 -440046.029}
SPL {X  -159.990, Y  +515.568, Z    +0.000, E1  +338.084, E3 -440061.259}
ENDSPLINE

SPLINE
SPL {X  -159.990, Y  +518.374, Z    +0.000, E1  +341.240, E3 -440073.846}
ENDSPLINE

SPLINE
SPL {X  -159.990, Y  +513.606, Z    +0.000, E1  +339.879, E3 -440089.757}
SPL {X  -159.990, Y  +508.660, Z    +0.000, E1  +338.515, E3 -440105.186}
SPL {X  -159.990, Y  +505.237, Z    +0.000, E1  +337.606, E3 -440115.444}
SPL {X  -159.990, Y  +501.963, Z    +0.000, E1  +336.712, E3 -440124.547}
SPL {X  -159.990, Y  +498.406, Z    +0.000, E1  +335.789, E3 -440134.298}
SPL {X  -159.990, Y  +494.693, Z    +0.000, E1  +334.929, E3 -440144.766}
SPL {X  -159.990, Y  +491.649, Z    +0.000, E1  +334.596, E3 -440155.968}
SPL {X  -159.990, Y  +488.807, Z    +0.000, E1  +334.603, E3 -440168.693}
SPL {X  -159.990, Y  +486.070, Z    +0.000, E1  +334.601, E3 -440180.924}
SPL {X  -159.990, Y  +483.747, Z    +0.000, E1  +334.616, E3 -440191.336}
SPL {X  -159.990, Y  +481.980, Z    +0.000, E1  +334.616, E3 -440199.234}
SPL {X  -159.990, Y  +479.252, Z    +0.000, E1  +334.588, E3 -440211.376}
SPL {X  -159.990, Y  +475.940, Z    +0.000, E1  +334.597, E3 -440226.196}
SPL {X  -159.990, Y  +473.026, Z    +0.000, E1  +334.601, E3 -440239.226}
SPL {X  -159.990, Y  +470.047, Z    +0.000, E1  +334.598, E3 -440252.544}
SPL {X  -159.990, Y  +466.213, Z    +0.000, E1  +334.567, E3 -440269.624}
SPL {X  -159.990, Y  +462.520, Z    +0.000, E1  +334.600, E3 -440286.192}
SPL {X  -159.990, Y  +460.081, Z    +0.000, E1  +334.610, E3 -440297.094}
SPL {X  -159.990, Y  +457.497, Z    +0.000, E1  +334.597, E3 -440308.618}
SPL {X  -159.990, Y  +455.126, Z    +0.000, E1  +334.611, E3 -440319.227}
SPL {X  -159.990, Y  +452.123, Z    +0.000, E1  +334.574, E3 -440332.584}
SPL {X  -159.990, Y  +448.503, Z    +0.000, E1  +334.590, E3 -440348.786}
SPL {X  -159.990, Y  +445.882, Z    +0.000, E1  +334.615, E3 -440360.588}
SPL {X  -159.990, Y  +443.345, Z    +0.000, E1  +334.610, E3 -440371.971}
SPL {X  -159.990, Y  +441.077, Z    +0.000, E1  +334.631, E3 -440382.169}
SPL {X  -159.990, Y  +438.608, Z    +0.000, E1  +334.608, E3 -440393.166}
SPL {X  -159.990, Y  +435.579, Z    +0.000, E1  +334.614, E3 -440406.720}
SPL {X  -159.990, Y  +432.613, Z    +0.000, E1  +334.610, E3 -440419.987}
SPL {X  -159.990, Y  +429.079, Z    +0.000, E1  +334.593, E3 -440435.758}
SPL {X  -159.990, Y  +426.149, Z    +0.000, E1  +334.626, E3 -440448.920}
SPL {X  -159.990, Y  +423.417, Z    +0.000, E1  +334.600, E3 -440461.085}
SPL {X  -159.990, Y  +419.467, Z    +0.000, E1  +334.583, E3 -440478.720}
SPL {X  -159.990, Y  +416.355, Z    +0.000, E1  +334.625, E3 -440492.717}
SPL {X  -159.990, Y  +413.684, Z    +0.000, E1  +334.603, E3 -440504.624}
SPL {X  -159.990, Y  +410.645, Z    +0.000, E1  +334.615, E3 -440518.236}
SPL {X  -159.990, Y  +408.351, Z    +0.000, E1  +334.628, E3 -440528.522}
SPL {X  -159.990, Y  +406.574, Z    +0.000, E1  +334.625, E3 -440536.439}
SPL {X  -159.990, Y  +404.255, Z    +0.000, E1  +334.609, E3 -440546.775}
SPL {X  -159.990, Y  +401.103, Z    +0.000, E1  +334.596, E3 -440560.839}
SPL {X  -159.990, Y  +398.389, Z    +0.000, E1  +334.619, E3 -440573.035}
SPL {X  -159.990, Y  +395.411, Z    +0.000, E1  +334.600, E3 -440586.332}
SPL {X  -159.990, Y  +392.473, Z    +0.000, E1  +334.623, E3 -440599.517}
SPL {X  -159.990, Y  +390.187, Z    +0.000, E1  +334.622, E3 -440609.775}
SPL {X  -159.990, Y  +387.503, Z    +0.000, E1  +334.622, E3 -440621.770}
SPL {X  -159.990, Y  +384.711, Z    +0.000, E1  +334.612, E3 -440634.214}
SPL {X  -159.988, Y  +381.794, Z    +0.000, E1  +334.611, E3 -440647.249}
SPL {X  -159.958, Y  +379.279, Z    +0.000, E1  +334.625, E3 -440658.539}
SPL {X  -159.867, Y  +376.223, Z    +0.000, E1  +334.608, E3 -440672.254}
SPL {X  -159.727, Y  +373.325, Z    +0.000, E1  +334.659, E3 -440685.418}
SPL {X  -159.549, Y  +370.634, Z    +0.000, E1  +334.653, E3 -440697.592}
SPL {X  -159.201, Y  +366.633, Z    +0.000, E1  +334.686, E3 -440715.784}
SPL {X  -158.798, Y  +363.007, Z    +0.000, E1  +334.761, E3 -440732.441}
SPL {X  -158.453, Y  +360.380, Z    +0.000, E1  +334.828, E3 -440744.586}
SPL {X  -158.127, Y  +358.155, Z    +0.000, E1  +334.874, E3 -440754.917}
SPL {X  -158.095, Y  +357.947, Z    +0.000, E1  +338.259, E3 -440786.489}
ENDSPLINE

SPLINE
SPL {X  -158.454, Y  +360.384, Z    +0.000, E1  +340.634, E3 -440798.640}
SPL {X  -159.737, Y  +373.507, Z    +0.000, E1  +349.689, E3 -440820.675}
SPL {X  -159.990, Y  +382.574, Z    +0.000, E1  +355.537, E3 -440827.363}
SPL {X  -159.990, Y  +387.496, Z    +0.000, E1  +358.996, E3 -440830.108}
SPL {X  -159.990, Y  +395.121, Z    +0.000, E1  +364.514, E3 -440834.421}
SPL {X  -159.990, Y  +407.941, Z    +0.000, E1  +374.126, E3 -440846.495}
SPL {X  -159.990, Y  +418.671, Z    +0.000, E1  +379.855, E3 -440865.911}
SPL {X  -159.990, Y  +429.878, Z    +0.000, E1  +383.330, E3 -440895.966}
SPL {X  -159.990, Y  +432.766, Z    +0.000, E1  +383.321, E3 -440910.189}
SPL {X  -159.990, Y  +434.794, Z    +0.000, E1  +383.304, E3 -440920.220}
SPL {X  -159.990, Y  +437.007, Z    +0.000, E1  +383.323, E3 -440931.072}
SPL {X  -159.990, Y  +439.778, Z    +0.000, E1  +383.323, E3 -440944.705}
SPL {X  -159.990, Y  +442.010, Z    +0.000, E1  +383.308, E3 -440955.726}
SPL {X  -159.990, Y  +443.729, Z    +0.000, E1  +383.310, E3 -440964.182}
SPL {X  -159.990, Y  +446.037, Z    +0.000, E1  +383.324, E3 -440975.519}
SPL {X  -159.990, Y  +448.341, Z    +0.000, E1  +383.317, E3 -440986.837}
SPL {X  -159.990, Y  +450.345, Z    +0.000, E1  +383.316, E3 -440996.715}
SPL {X  -159.990, Y  +452.828, Z    +0.000, E1  +383.330, E3 -441008.914}
SPL {X  -159.990, Y  +456.338, Z    +0.000, E1  +383.359, E3 -441026.106}
SPL {X  -159.990, Y  +459.480, Z    +0.000, E1  +383.323, E3 -441041.647}
SPL {X  -159.990, Y  +461.803, Z    +0.000, E1  +383.322, E3 -441053.083}
SPL {X  -159.990, Y  +464.971, Z    +0.000, E1  +383.357, E3 -441068.589}
SPL {X  -159.990, Y  +467.934, Z    +0.000, E1  +383.321, E3 -441083.246}
SPL {X  -159.990, Y  +469.939, Z    +0.000, E1  +383.319, E3 -441093.108}
SPL {X  -159.990, Y  +472.144, Z    +0.000, E1  +383.327, E3 -441103.958}
SPL {X  -159.990, Y  +474.152, Z    +0.000, E1  +383.309, E3 -441113.910}
SPL {X  -159.990, Y  +476.560, Z    +0.000, E1  +383.332, E3 -441125.718}
SPL {X  -159.990, Y  +478.770, Z    +0.000, E1  +383.306, E3 -441136.644}
SPL {X  -159.990, Y  +480.905, Z    +0.000, E1  +383.327, E3 -441147.112}
SPL {X  -159.990, Y  +484.251, Z    +0.000, E1  +383.352, E3 -441163.527}
SPL {X  -159.990, Y  +488.031, Z    +0.000, E1  +383.345, E3 -441182.160}
SPL {X  -159.990, Y  +491.121, Z    +0.000, E1  +383.323, E3 -441197.406}
SPL {X  -159.990, Y  +493.610, Z    +0.000, E1  +383.323, E3 -441209.659}
SPL {X  -159.990, Y  +496.863, Z    +0.000, E1  +383.350, E3 -441225.619}
SPL {X  -159.990, Y  +499.995, Z    +0.000, E1  +383.324, E3 -441241.080}
SPL {X  -159.990, Y  +502.341, Z    +0.000, E1  +383.320, E3 -441252.639}
SPL {X  -159.990, Y  +504.419, Z    +0.000, E1  +383.313, E3 -441262.881}
SPL {X  -159.990, Y  +507.187, Z    +0.000, E1  +383.346, E3 -441276.434}
SPL {X  -159.990, Y  +510.344, Z    +0.000, E1  +383.327, E3 -441292.019}
SPL {X  -159.990, Y  +512.484, Z    +0.000, E1  +383.309, E3 -441302.591}
SPL {X  -159.990, Y  +514.016, Z    +0.000, E1  +383.308, E3 -441310.140}
SPL {X  -159.990, Y  +516.195, Z    +0.000, E1  +383.325, E3 -441320.828}
SPL {X  -159.990, Y  +518.925, Z    +0.000, E1  +383.333, E3 -441334.191}
SPL {X  -159.990, Y  +521.408, Z    +0.000, E1  +383.329, E3 -441346.400}
SPL {X  -159.990, Y  +523.942, Z    +0.000, E1  +383.333, E3 -441358.893}
SPL {X  -159.990, Y  +527.007, Z    +0.000, E1  +383.339, E3 -441373.992}
SPL {X  -159.990, Y  +529.993, Z    +0.000, E1  +383.329, E3 -441388.695}
SPL {X  -159.990, Y  +532.441, Z    +0.000, E1  +383.322, E3 -441400.745}
SPL {X  -159.990, Y  +534.618, Z    +0.000, E1  +383.322, E3 -441411.478}
SPL {X  -159.990, Y  +537.024, Z    +0.000, E1  +383.321, E3 -441423.341}
SPL {X  -159.990, Y  +539.129, Z    +0.000, E1  +383.310, E3 -441433.724}
SPL {X  -159.990, Y  +541.183, Z    +0.000, E1  +383.319, E3 -441443.821}
SPL {X  -159.990, Y  +543.647, Z    +0.000, E1  +383.325, E3 -441455.924}
SPL {X  -159.990, Y  +546.832, Z    +0.000, E1  +383.349, E3 -441471.546}
SPL {X  -159.990, Y  +549.756, Z    +0.000, E1  +383.320, E3 -441485.987}
SPL {X  -159.990, Y  +551.655, Z    +0.000, E1  +383.320, E3 -441495.338}
SPL {X  -159.990, Y  +553.711, Z    +0.000, E1  +383.317, E3 -441505.460}
SPL {X  -159.990, Y  +556.481, Z    +0.000, E1  +383.354, E3 -441519.022}
SPL {X  -159.990, Y  +559.475, Z    +0.000, E1  +383.321, E3 -441533.827}
SPL {X  -159.990, Y  +561.830, Z    +0.000, E1  +383.325, E3 -441545.412}
SPL {X  -159.990, Y  +564.273, Z    +0.000, E1  +383.325, E3 -441557.436}
SPL {X  -159.990, Y  +566.342, Z    +0.000, E1  +383.314, E3 -441567.640}
SPL {X  -159.990, Y  +568.184, Z    +0.000, E1  +383.317, E3 -441576.701}
SPL {X  -159.990, Y  +570.314, Z    +0.000, E1  +383.326, E3 -441587.164}
SPL {X  -159.990, Y  +573.444, Z    +0.000, E1  +383.356, E3 -441602.503}
SPL {X  -159.990, Y  +577.161, Z    +0.000, E1  +383.346, E3 -441620.827}
SPL {X  -159.990, Y  +580.840, Z    +0.000, E1  +383.355, E3 -441638.877}
SPL {X  -159.990, Y  +583.973, Z    +0.000, E1  +383.332, E3 -441654.338}
SPL {X  -159.990, Y  +586.020, Z    +0.000, E1  +383.323, E3 -441664.422}
SPL {X  -159.990, Y  +587.711, Z    +0.000, E1  +383.318, E3 -441672.762}
SPL {X  -159.990, Y  +589.763, Z    +0.000, E1  +383.328, E3 -441682.838}
SPL {X  -159.990, Y  +591.698, Z    +0.000, E1  +383.324, E3 -441692.323}
SPL {X  -159.990, Y  +593.847, Z    +0.000, E1  +383.340, E3 -441702.853}
SPL {X  -159.990, Y  +597.018, Z    +0.000, E1  +383.367, E3 -441718.385}
SPL {X  -159.990, Y  +599.887, Z    +0.000, E1  +383.341, E3 -441732.489}
SPL {X  -159.990, Y  +601.949, Z    +0.000, E1  +383.344, E3 -441742.616}
SPL {X  -159.990, Y  +605.106, Z    +0.000, E1  +383.383, E3 -441758.062}
SPL {X  -159.990, Y  +608.111, Z    +0.000, E1  +383.342, E3 -441772.913}
SPL {X  -159.990, Y  +610.073, Z    +0.000, E1  +383.343, E3 -441782.571}
SPL {X  -159.990, Y  +612.330, Z    +0.000, E1  +383.340, E3 -441793.699}
SPL {X  -159.990, Y  +615.036, Z    +0.000, E1  +383.353, E3 -441806.986}
SPL {X  -159.990, Y  +618.481, Z    +0.000, E1  +383.366, E3 -441823.924}
SPL {X  -159.990, Y  +621.517, Z    +0.000, E1  +383.337, E3 -441838.907}
SPL {X  -159.990, Y  +623.764, Z    +0.000, E1  +383.335, E3 -441849.957}
SPL {X  -159.990, Y  +626.608, Z    +0.000, E1  +383.361, E3 -441863.882}
SPL {X  -159.990, Y  +630.271, Z    +0.000, E1  +383.375, E3 -441881.844}
SPL {X  -159.990, Y  +633.318, Z    +0.000, E1  +383.339, E3 -441896.921}
SPL {X  -159.990, Y  +635.650, Z    +0.000, E1  +383.339, E3 -441908.392}
SPL {X  -159.990, Y  +638.406, Z    +0.000, E1  +383.354, E3 -441921.959}
SPL {X  -159.990, Y  +641.131, Z    +0.000, E1  +383.320, E3 -441935.483}
SPL {X  -159.990, Y  +644.241, Z    +0.000, E1  +383.355, E3 -441950.761}
SPL {X  -159.990, Y  +648.287, Z    +0.000, E1  +383.349, E3 -441970.718}
SPL {X  -159.990, Y  +651.427, Z    +0.000, E1  +383.319, E3 -441986.213}
SPL {X  -159.990, Y  +653.536, Z    +0.000, E1  +383.313, E3 -441996.594}
SPL {X  -159.990, Y  +656.380, Z    +0.000, E1  +383.347, E3 -442010.530}
SPL {X  -159.990, Y  +659.180, Z    +0.000, E1  +383.314, E3 -442024.378}
SPL {X  -159.990, Y  +661.392, Z    +0.000, E1  +383.318, E3 -442035.272}
SPL {X  -159.990, Y  +663.662, Z    +0.000, E1  +383.322, E3 -442046.396}
SPL {X  -159.990, Y  +665.964, Z    +0.000, E1  +383.328, E3 -442057.686}
SPL {X  -159.990, Y  +668.989, Z    +0.000, E1  +383.359, E3 -442072.522}
SPL {X  -159.983, Y  +672.946, Z    +0.000, E1  +383.359, E3 -442092.004}
SPL {X  -159.924, Y  +676.110, Z    +0.000, E1  +383.320, E3 -442107.703}
SPL {X  -159.801, Y  +679.265, Z    +0.000, E1  +383.327, E3 -442123.321}
SPL {X  -159.626, Y  +682.287, Z    +0.000, E1  +383.280, E3 -442138.420}
SPL {X  -159.462, Y  +684.486, Z    +0.000, E1  +383.258, E3 -442149.419}
SPL {X  -159.289, Y  +686.457, Z    +0.000, E1  +383.223, E3 -442159.330}
SPL {X  -159.052, Y  +688.801, Z    +0.000, E1  +383.217, E3 -442171.064}
SPL {X  -158.770, Y  +691.222, Z    +0.000, E1  +383.158, E3 -442183.322}
SPL {X  -158.553, Y  +692.896, Z    +0.000, E1  +383.130, E3 -442191.787}
ENDSPLINE

SPLINE
SPL {X  -158.898, Y  +690.164, Z    +0.000, E1  +378.236, E3 -442225.143}
SPL {X  -159.149, Y  +687.882, Z    +0.000, E1  +376.368, E3 -442232.431}
SPL {X  -159.957, Y  +674.769, Z    +0.000, E1  +367.092, E3 -442252.290}
SPL {X  -159.990, Y  +671.516, Z    +0.000, E1  +364.944, E3 -442254.676}
SPL {X  -159.990, Y  +663.928, Z    +0.000, E1  +359.662, E3 -442259.768}
SPL {X  -159.990, Y  +658.009, Z    +0.000, E1  +355.226, E3 -442263.468}
SPL {X  -159.990, Y  +651.879, Z    +0.000, E1  +350.548, E3 -442268.530}
SPL {X  -159.990, Y  +637.832, Z    +0.000, E1  +341.694, E3 -442286.121}
SPL {X  -159.990, Y  +626.634, Z    +0.000, E1  +337.968, E3 -442316.974}
SPL {X  -159.990, Y  +624.622, Z    +0.000, E1  +337.980, E3 -442327.558}
SPL {X  -159.990, Y  +622.489, Z    +0.000, E1  +337.969, E3 -442338.724}
SPL {X  -159.990, Y  +619.955, Z    +0.000, E1  +337.968, E3 -442352.014}
SPL {X  -159.990, Y  +617.386, Z    +0.000, E1  +337.968, E3 -442365.489}
SPL {X  -159.990, Y  +614.863, Z    +0.000, E1  +337.969, E3 -442378.721}
SPL {X  -159.990, Y  +612.600, Z    +0.000, E1  +337.975, E3 -442390.605}
SPL {X  -159.990, Y  +610.646, Z    +0.000, E1  +337.979, E3 -442400.863}
SPL {X  -159.990, Y  +608.810, Z    +0.000, E1  +337.977, E3 -442410.496}
SPL {X  -159.990, Y  +606.481, Z    +0.000, E1  +337.967, E3 -442422.671}
SPL {X  -159.990, Y  +603.419, Z    +0.000, E1  +337.936, E3 -442438.611}
SPL {X  -159.990, Y  +600.642, Z    +0.000, E1  +337.968, E3 -442453.240}
SPL {X  -159.990, Y  +598.568, Z    +0.000, E1  +337.954, E3 -442464.033}
SPL {X  -159.990, Y  +595.493, Z    +0.000, E1  +337.930, E3 -442480.116}
SPL {X  -159.990, Y  +592.865, Z    +0.000, E1  +337.964, E3 -442493.945}
SPL {X  -159.990, Y  +590.803, Z    +0.000, E1  +337.954, E3 -442504.735}
SPL {X  -159.990, Y  +588.288, Z    +0.000, E1  +337.950, E3 -442517.900}
SPL {X  -159.990, Y  +586.040, Z    +0.000, E1  +337.954, E3 -442529.645}
SPL {X  -159.990, Y  +584.080, Z    +0.000, E1  +337.953, E3 -442539.905}
SPL {X  -159.990, Y  +581.924, Z    +0.000, E1  +337.949, E3 -442551.205}
SPL {X  -159.990, Y  +579.673, Z    +0.000, E1  +337.950, E3 -442563.003}
SPL {X  -159.990, Y  +576.961, Z    +0.000, E1  +337.936, E3 -442577.183}
SPL {X  -159.990, Y  +574.188, Z    +0.000, E1  +337.947, E3 -442591.730}
SPL {X  -159.990, Y  +571.954, Z    +0.000, E1  +337.959, E3 -442603.487}
SPL {X  -159.990, Y  +570.110, Z    +0.000, E1  +337.958, E3 -442613.138}
SPL {X  -159.990, Y  +568.165, Z    +0.000, E1  +337.957, E3 -442623.318}
SPL {X  -159.990, Y  +565.292, Z    +0.000, E1  +337.922, E3 -442638.296}
SPL {X  -159.990, Y  +562.598, Z    +0.000, E1  +337.958, E3 -442652.507}
SPL {X  -159.990, Y  +560.652, Z    +0.000, E1  +337.962, E3 -442662.719}
SPL {X  -159.990, Y  +558.143, Z    +0.000, E1  +337.928, E3 -442675.751}
SPL {X  -159.990, Y  +555.329, Z    +0.000, E1  +337.943, E3 -442690.495}
SPL {X  -159.990, Y  +553.115, Z    +0.000, E1  +337.946, E3 -442702.100}
SPL {X  -159.990, Y  +550.886, Z    +0.000, E1  +337.944, E3 -442713.782}
SPL {X  -159.990, Y  +548.568, Z    +0.000, E1  +337.944, E3 -442725.903}
SPL {X  -159.990, Y  +545.859, Z    +0.000, E1  +337.926, E3 -442740.052}
SPL {X  -159.990, Y  +542.390, Z    +0.000, E1  +337.914, E3 -442758.223}
SPL {X  -159.990, Y  +539.341, Z    +0.000, E1  +337.944, E3 -442774.244}
SPL {X  -159.990, Y  +536.935, Z    +0.000, E1  +337.942, E3 -442786.834}
SPL {X  -159.990, Y  +534.656, Z    +0.000, E1  +337.946, E3 -442798.778}
SPL {X  -159.990, Y  +532.453, Z    +0.000, E1  +337.944, E3 -442810.305}
SPL {X  -159.990, Y  +530.660, Z    +0.000, E1  +337.952, E3 -442819.707}
SPL {X  -159.990, Y  +528.702, Z    +0.000, E1  +337.939, E3 -442829.920}
SPL {X  -159.990, Y  +525.760, Z    +0.000, E1  +337.914, E3 -442845.262}
SPL {X  -159.990, Y  +522.838, Z    +0.000, E1  +337.933, E3 -442860.628}
SPL {X  -159.990, Y  +520.708, Z    +0.000, E1  +337.953, E3 -442871.822}
SPL {X  -159.990, Y  +518.216, Z    +0.000, E1  +337.909, E3 -442884.739}
SPL {X  -159.990, Y  +515.568, Z    +0.000, E1  +338.084, E3 -442899.968}
ENDSPLINE

SPLINE
SPL {X  -159.990, Y  +518.374, Z    +0.000, E1  +341.240, E3 -442912.556}
ENDSPLINE

SPLINE
SPL {X  -159.990, Y  +513.606, Z    +0.000, E1  +339.879, E3 -442928.467}
SPL {X  -159.990, Y  +508.660, Z    +0.000, E1  +338.515, E3 -442943.896}
SPL {X  -159.990, Y  +505.237, Z    +0.000, E1  +337.606, E3 -442954.153}
SPL {X  -159.990, Y  +501.963, Z    +0.000, E1  +336.712, E3 -442963.257}
SPL {X  -159.990, Y  +498.406, Z    +0.000, E1  +335.789, E3 -442973.008}
SPL {X  -159.990, Y  +494.693, Z    +0.000, E1  +334.929, E3 -442983.475}
SPL {X  -159.990, Y  +491.649, Z    +0.000, E1  +334.596, E3 -442994.678}
SPL {X  -159.990, Y  +488.807, Z    +0.000, E1  +334.603, E3 -443007.402}
SPL {X  -159.990, Y  +486.070, Z    +0.000, E1  +334.601, E3 -443019.633}
SPL {X  -159.990, Y  +483.747, Z    +0.000, E1  +334.616, E3 -443030.046}
SPL {X  -159.990, Y  +481.980, Z    +0.000, E1  +334.616, E3 -443037.944}
SPL {X  -159.990, Y  +479.252, Z    +0.000, E1  +334.588, E3 -443050.086}
SPL {X  -159.990, Y  +475.940, Z    +0.000, E1  +334.597, E3 -443064.906}
SPL {X  -159.990, Y  +473.026, Z    +0.000, E1  +334.601, E3 -443077.935}
SPL {X  -159.990, Y  +470.047, Z    +0.000, E1  +334.598, E3 -443091.254}
SPL {X  -159.990, Y  +466.213, Z    +0.000, E1  +334.567, E3 -443108.334}
SPL {X  -159.990, Y  +462.520, Z    +0.000, E1  +334.600, E3 -443124.902}
SPL {X  -159.990, Y  +460.081, Z    +0.000, E1  +334.610, E3 -443135.804}
SPL {X  -159.990, Y  +457.497, Z    +0.000, E1  +334.597, E3 -443147.328}
SPL {X  -159.990, Y  +455.126, Z    +0.000, E1  +334.611, E3 -443157.936}
SPL {X  -159.990, Y  +452.123, Z    +0.000, E1  +334.574, E3 -443171.294}
SPL {X  -159.990, Y  +448.503, Z    +0.000, E1  +334.590, E3 -443187.496}
SPL {X  -159.990, Y  +445.882, Z    +0.000, E1  +334.615, E3 -443199.298}
SPL {X  -159.990, Y  +443.345, Z    +0.000, E1  +334.610, E3 -443210.680}
SPL {X  -159.990, Y  +441.077, Z    +0.000, E1  +334.631, E3 -443220.879}
SPL {X  -159.990, Y  +438.608, Z    +0.000, E1  +334.608, E3 -443231.875}
SPL {X  -159.990, Y  +434.852, Z    +0.000, E1  +334.585, E3 -443248.630}
SPL {X  -159.990, Y  +430.645, Z    +0.000, E1  +334.586, E3 -443267.449}
SPL {X  -159.990, Y  +426.865, Z    +0.000, E1  +334.602, E3 -443284.379}
SPL {X  -159.990, Y  +424.251, Z    +0.000, E1  +334.625, E3 -443296.116}
SPL {X  -159.990, Y  +421.010, Z    +0.000, E1  +334.582, E3 -443310.531}
SPL {X  -159.990, Y  +417.103, Z    +0.000, E1  +334.600, E3 -443328.034}
SPL {X  -159.990, Y  +413.684, Z    +0.000, E1  +334.603, E3 -443343.334}
SPL {X  -159.990, Y  +410.645, Z    +0.000, E1  +334.615, E3 -443356.946}
SPL {X  -159.990, Y  +407.450, Z    +0.000, E1  +334.599, E3 -443371.194}
SPL {X  -159.990, Y  +403.513, Z    +0.000, E1  +334.580, E3 -443388.747}
SPL {X  -159.990, Y  +399.294, Z    +0.000, E1  +334.582, E3 -443407.627}
SPL {X  -159.990, Y  +395.411, Z    +0.000, E1  +334.600, E3 -443425.042}
SPL {X  -159.990, Y  +392.473, Z    +0.000, E1  +334.623, E3 -443438.227}
SPL {X  -159.990, Y  +390.187, Z    +0.000, E1  +334.622, E3 -443448.485}
SPL {X  -159.990, Y  +387.503, Z    +0.000, E1  +334.622, E3 -443460.480}
SPL {X  -159.990, Y  +384.711, Z    +0.000, E1  +334.612, E3 -443472.924}
SPL {X  -159.988, Y  +381.794, Z    +0.000, E1  +334.611, E3 -443485.958}
SPL {X  -159.958, Y  +379.279, Z    +0.000, E1  +334.625, E3 -443497.249}
SPL {X  -159.867, Y  +376.223, Z    +0.000, E1  +334.608, E3 -443510.963}
SPL {X  -159.659, Y  +372.220, Z    +0.000, E1  +334.632, E3 -443529.085}
SPL {X  -159.379, Y  +368.534, Z    +0.000, E1  +334.684, E3 -443545.871}
SPL {X  -159.113, Y  +365.767, Z    +0.000, E1  +334.734, E3 -443558.511}
SPL {X  -158.798, Y  +363.007, Z    +0.000, E1  +334.761, E3 -443571.151}
SPL {X  -158.453, Y  +360.380, Z    +0.000, E1  +334.828, E3 -443583.296}
SPL {X  -158.127, Y  +358.155, Z    +0.000, E1  +334.874, E3 -443593.626}
SPL {X  -158.095, Y  +357.947, Z    +0.000, E1  +338.259, E3 -443625.199}
ENDSPLINE

SPLINE
SPL {X  -158.454, Y  +360.384, Z    +0.000, E1  +340.634, E3 -443637.350}
SPL {X  -159.737, Y  +373.507, Z    +0.000, E1  +349.689, E3 -443659.385}
SPL {X  -159.990, Y  +382.574, Z    +0.000, E1  +355.537, E3 -443666.073}
SPL {X  -159.990, Y  +387.496, Z    +0.000, E1  +358.996, E3 -443668.818}
SPL {X  -159.990, Y  +395.121, Z    +0.000, E1  +364.514, E3 -443673.130}
SPL {X  -159.990, Y  +407.941, Z    +0.000, E1  +374.126, E3 -443685.205}
SPL {X  -159.990, Y  +418.671, Z    +0.000, E1  +379.855, E3 -443704.621}
SPL {X  -159.990, Y  +428.534, Z    +0.000, E1  +383.299, E3 -443728.141}
SPL {X  -159.990, Y  +430.313, Z    +0.000, E1  +383.313, E3 -443736.854}
SPL {X  -159.990, Y  +432.766, Z    +0.000, E1  +383.321, E3 -443748.898}
SPL {X  -159.990, Y  +434.794, Z    +0.000, E1  +383.304, E3 -443758.930}
SPL {X  -159.990, Y  +437.007, Z    +0.000, E1  +383.323, E3 -443769.782}
SPL {X  -159.990, Y  +439.778, Z    +0.000, E1  +383.323, E3 -443783.414}
SPL {X  -159.990, Y  +442.010, Z    +0.000, E1  +383.308, E3 -443794.435}
SPL {X  -159.990, Y  +443.729, Z    +0.000, E1  +383.310, E3 -443802.892}
SPL {X  -159.990, Y  +446.037, Z    +0.000, E1  +383.324, E3 -443814.229}
SPL {X  -159.990, Y  +448.341, Z    +0.000, E1  +383.317, E3 -443825.546}
SPL {X  -159.990, Y  +450.345, Z    +0.000, E1  +383.316, E3 -443835.424}
SPL {X  -159.990, Y  +452.828, Z    +0.000, E1  +383.330, E3 -443847.624}
SPL {X  -159.990, Y  +456.338, Z    +0.000, E1  +383.359, E3 -443864.816}
SPL {X  -159.990, Y  +459.480, Z    +0.000, E1  +383.323, E3 -443880.357}
SPL {X  -159.990, Y  +461.803, Z    +0.000, E1  +383.322, E3 -443891.792}
SPL {X  -159.990, Y  +464.971, Z    +0.000, E1  +383.357, E3 -443907.298}
SPL {X  -159.990, Y  +467.934, Z    +0.000, E1  +383.321, E3 -443921.956}
SPL {X  -159.990, Y  +469.939, Z    +0.000, E1  +383.319, E3 -443931.817}
SPL {X  -159.990, Y  +472.144, Z    +0.000, E1  +383.327, E3 -443942.668}
SPL {X  -159.990, Y  +474.152, Z    +0.000, E1  +383.309, E3 -443952.620}
SPL {X  -159.990, Y  +475.762, Z    +0.000, E1  +383.308, E3 -443960.549}
SPL {X  -159.990, Y  +478.041, Z    +0.000, E1  +383.328, E3 -443971.725}
SPL {X  -159.990, Y  +480.905, Z    +0.000, E1  +383.327, E3 -443985.821}
SPL {X  -159.990, Y  +484.251, Z    +0.000, E1  +383.352, E3 -444002.237}
SPL {X  -159.990, Y  +488.031, Z    +0.000, E1  +383.345, E3 -444020.870}
SPL {X  -159.990, Y  +491.121, Z    +0.000, E1  +383.323, E3 -444036.115}
SPL {X  -159.990, Y  +493.610, Z    +0.000, E1  +383.323, E3 -444048.368}
SPL {X  -159.990, Y  +496.863, Z    +0.000, E1  +383.350, E3 -444064.328}
SPL {X  -159.990, Y  +499.995, Z    +0.000, E1  +383.324, E3 -444079.790}
SPL {X  -159.990, Y  +502.341, Z    +0.000, E1  +383.320, E3 -444091.349}
SPL {X  -159.990, Y  +505.377, Z    +0.000, E1  +383.346, E3 -444106.239}
SPL {X  -159.990, Y  +508.024, Z    +0.000, E1  +383.315, E3 -444119.322}
SPL {X  -159.990, Y  +510.344, Z    +0.000, E1  +383.327, E3 -444130.728}
SPL {X  -159.990, Y  +513.289, Z    +0.000, E1  +383.332, E3 -444145.218}
SPL {X  -159.990, Y  +516.195, Z    +0.000, E1  +383.325, E3 -444159.537}
SPL {X  -159.990, Y  +518.925, Z    +0.000, E1  +383.333, E3 -444172.901}
SPL {X  -159.990, Y  +521.408, Z    +0.000, E1  +383.329, E3 -444185.110}
SPL {X  -159.990, Y  +523.942, Z    +0.000, E1  +383.333, E3 -444197.602}
SPL {X  -159.990, Y  +526.221, Z    +0.000, E1  +383.314, E3 -444208.878}
SPL {X  -159.990, Y  +527.834, Z    +0.000, E1  +383.311, E3 -444216.828}
SPL {X  -159.990, Y  +529.993, Z    +0.000, E1  +383.329, E3 -444227.404}
SPL {X  -159.990, Y  +532.441, Z    +0.000, E1  +383.322, E3 -444239.455}
SPL {X  -159.990, Y  +534.618, Z    +0.000, E1  +383.322, E3 -444250.188}
SPL {X  -159.990, Y  +537.024, Z    +0.000, E1  +383.321, E3 -444262.051}
SPL {X  -159.990, Y  +539.129, Z    +0.000, E1  +383.310, E3 -444272.433}
SPL {X  -159.990, Y  +541.183, Z    +0.000, E1  +383.319, E3 -444282.530}
SPL {X  -159.990, Y  +543.647, Z    +0.000, E1  +383.325, E3 -444294.633}
SPL {X  -159.990, Y  +546.832, Z    +0.000, E1  +383.349, E3 -444310.256}
SPL {X  -159.990, Y  +549.756, Z    +0.000, E1  +383.320, E3 -444324.697}
SPL {X  -159.990, Y  +551.655, Z    +0.000, E1  +383.320, E3 -444334.048}
SPL {X  -159.990, Y  +553.711, Z    +0.000, E1  +383.317, E3 -444344.170}
SPL {X  -159.990, Y  +555.637, Z    +0.000, E1  +383.323, E3 -444353.639}
SPL {X  -159.990, Y  +558.758, Z    +0.000, E1  +383.351, E3 -444368.948}
SPL {X  -159.990, Y  +561.830, Z    +0.000, E1  +383.325, E3 -444384.121}
SPL {X  -159.990, Y  +564.273, Z    +0.000, E1  +383.325, E3 -444396.146}
SPL {X  -159.990, Y  +567.351, Z    +0.000, E1  +383.348, E3 -444411.242}
SPL {X  -159.990, Y  +570.314, Z    +0.000, E1  +383.326, E3 -444425.874}
SPL {X  -159.990, Y  +572.504, Z    +0.000, E1  +383.321, E3 -444436.658}
SPL {X  -159.990, Y  +575.653, Z    +0.000, E1  +383.355, E3 -444452.095}
SPL {X  -159.990, Y  +578.932, Z    +0.000, E1  +383.330, E3 -444468.278}
SPL {X  -159.990, Y  +581.497, Z    +0.000, E1  +383.329, E3 -444480.863}
SPL {X  -159.990, Y  +583.973, Z    +0.000, E1  +383.332, E3 -444493.048}
SPL {X  -159.990, Y  +586.020, Z    +0.000, E1  +383.323, E3 -444503.132}
SPL {X  -159.990, Y  +587.711, Z    +0.000, E1  +383.318, E3 -444511.471}
SPL {X  -159.990, Y  +589.763, Z    +0.000, E1  +383.328, E3 -444521.548}
SPL {X  -159.990, Y  +591.698, Z    +0.000, E1  +383.324, E3 -444531.032}
SPL {X  -159.990, Y  +593.847, Z    +0.000, E1  +383.340, E3 -444541.563}
SPL {X  -159.990, Y  +597.018, Z    +0.000, E1  +383.367, E3 -444557.095}
SPL {X  -159.990, Y  +599.887, Z    +0.000, E1  +383.341, E3 -444571.199}
SPL {X  -159.990, Y  +601.949, Z    +0.000, E1  +383.344, E3 -444581.326}
SPL {X  -159.990, Y  +605.106, Z    +0.000, E1  +383.383, E3 -444596.772}
SPL {X  -159.990, Y  +608.111, Z    +0.000, E1  +383.342, E3 -444611.623}
SPL {X  -159.990, Y  +610.073, Z    +0.000, E1  +383.343, E3 -444621.281}
SPL {X  -159.990, Y  +612.330, Z    +0.000, E1  +383.340, E3 -444632.408}
SPL {X  -159.990, Y  +615.036, Z    +0.000, E1  +383.353, E3 -444645.696}
SPL {X  -159.990, Y  +618.481, Z    +0.000, E1  +383.366, E3 -444662.634}
SPL {X  -159.990, Y  +621.517, Z    +0.000, E1  +383.337, E3 -444677.617}
SPL {X  -159.990, Y  +623.764, Z    +0.000, E1  +383.335, E3 -444688.667}
SPL {X  -159.990, Y  +626.608, Z    +0.000, E1  +383.361, E3 -444702.592}
SPL {X  -159.990, Y  +630.271, Z    +0.000, E1  +383.375, E3 -444720.553}
SPL {X  -159.990, Y  +633.318, Z    +0.000, E1  +383.339, E3 -444735.631}
SPL {X  -159.990, Y  +635.650, Z    +0.000, E1  +383.339, E3 -444747.102}
SPL {X  -159.990, Y  +638.406, Z    +0.000, E1  +383.354, E3 -444760.668}
SPL {X  -159.990, Y  +641.831, Z    +0.000, E1  +383.342, E3 -444777.616}
SPL {X  -159.990, Y  +644.884, Z    +0.000, E1  +383.324, E3 -444792.703}
SPL {X  -159.990, Y  +647.550, Z    +0.000, E1  +383.318, E3 -444805.869}
SPL {X  -159.990, Y  +650.790, Z    +0.000, E1  +383.346, E3 -444821.736}
SPL {X  -159.990, Y  +654.543, Z    +0.000, E1  +383.348, E3 -444840.189}
SPL {X  -159.990, Y  +658.319, Z    +0.000, E1  +383.349, E3 -444858.779}
SPL {X  -159.990, Y  +661.392, Z    +0.000, E1  +383.318, E3 -444873.982}
SPL {X  -159.990, Y  +663.662, Z    +0.000, E1  +383.322, E3 -444885.106}
SPL {X  -159.990, Y  +665.964, Z    +0.000, E1  +383.328, E3 -444896.396}
SPL {X  -159.990, Y  +667.870, Z    +0.000, E1  +383.320, E3 -444905.803}
SPL {X  -159.990, Y  +669.861, Z    +0.000, E1  +383.321, E3 -444915.604}
SPL {X  -159.990, Y  +671.893, Z    +0.000, E1  +383.319, E3 -444925.612}
SPL {X  -159.974, Y  +673.789, Z    +0.000, E1  +383.323, E3 -444934.928}
SPL {X  -159.924, Y  +676.110, Z    +0.000, E1  +383.320, E3 -444946.412}
SPL {X  -159.801, Y  +679.265, Z    +0.000, E1  +383.327, E3 -444962.031}
SPL {X  -159.626, Y  +682.287, Z    +0.000, E1  +383.280, E3 -444977.130}
SPL {X  -159.462, Y  +684.486, Z    +0.000, E1  +383.258, E3 -444988.129}
SPL {X  -159.212, Y  +687.262, Z    +0.000, E1  +383.238, E3 -445002.033}
SPL {X  -158.971, Y  +689.529, Z    +0.000, E1  +383.181, E3 -445013.493}
SPL {X  -158.658, Y  +692.098, Z    +0.000, E1  +383.176, E3 -445026.399}
ENDSPLINE

SPLINE
SPL {X  -159.063, Y  +688.696, Z    +0.000, E1  +377.094, E3 -445068.618}
SPL {X  -159.957, Y  +674.769, Z    +0.000, E1  +367.092, E3 -445091.000}
SPL {X  -159.990, Y  +671.516, Z    +0.000, E1  +364.944, E3 -445093.385}
SPL {X  -159.990, Y  +663.928, Z    +0.000, E1  +359.662, E3 -445098.477}
SPL {X  -159.990, Y  +658.009, Z    +0.000, E1  +355.226, E3 -445102.177}
SPL {X  -159.990, Y  +651.879, Z    +0.000, E1  +350.548, E3 -445107.240}
SPL {X  -159.990, Y  +637.832, Z    +0.000, E1  +341.694, E3 -445124.831}
SPL {X  -159.990, Y  +626.634, Z    +0.000, E1  +337.968, E3 -445155.684}
SPL {X  -159.990, Y  +624.622, Z    +0.000, E1  +337.980, E3 -445166.268}
SPL {X  -159.990, Y  +622.489, Z    +0.000, E1  +337.969, E3 -445177.434}
SPL {X  -159.990, Y  +619.955, Z    +0.000, E1  +337.968, E3 -445190.724}
SPL {X  -159.990, Y  +617.386, Z    +0.000, E1  +337.968, E3 -445204.199}
SPL {X  -159.990, Y  +614.863, Z    +0.000, E1  +337.969, E3 -445217.431}
SPL {X  -159.990, Y  +612.600, Z    +0.000, E1  +337.975, E3 -445229.315}
SPL {X  -159.990, Y  +610.646, Z    +0.000, E1  +337.979, E3 -445239.573}
SPL {X  -159.990, Y  +608.810, Z    +0.000, E1  +337.977, E3 -445249.205}
SPL {X  -159.990, Y  +605.804, Z    +0.000, E1  +337.936, E3 -445264.851}
SPL {X  -159.990, Y  +602.819, Z    +0.000, E1  +337.963, E3 -445280.522}
SPL {X  -159.990, Y  +600.642, Z    +0.000, E1  +337.968, E3 -445291.950}
SPL {X  -159.990, Y  +598.568, Z    +0.000, E1  +337.954, E3 -445302.743}
SPL {X  -159.990, Y  +595.493, Z    +0.000, E1  +337.930, E3 -445318.826}
SPL {X  -159.990, Y  +592.865, Z    +0.000, E1  +337.964, E3 -445332.654}
SPL {X  -159.990, Y  +590.803, Z    +0.000, E1  +337.954, E3 -445343.445}
SPL {X  -159.990, Y  +588.288, Z    +0.000, E1  +337.950, E3 -445356.609}
SPL {X  -159.990, Y  +586.040, Z    +0.000, E1  +337.954, E3 -445368.354}
SPL {X  -159.990, Y  +584.080, Z    +0.000, E1  +337.953, E3 -445378.614}
SPL {X  -159.990, Y  +581.924, Z    +0.000, E1  +337.949, E3 -445389.915}
SPL {X  -159.990, Y  +579.673, Z    +0.000, E1  +337.950, E3 -445401.713}
SPL {X  -159.990, Y  +576.961, Z    +0.000, E1  +337.936, E3 -445415.892}
SPL {X  -159.990, Y  +574.188, Z    +0.000, E1  +337.947, E3 -445430.440}
SPL {X  -159.990, Y  +571.954, Z    +0.000, E1  +337.959, E3 -445442.197}
SPL {X  -159.990, Y  +570.110, Z    +0.000, E1  +337.958, E3 -445451.848}
SPL {X  -159.990, Y  +568.165, Z    +0.000, E1  +337.957, E3 -445462.027}
SPL {X  -159.990, Y  +565.292, Z    +0.000, E1  +337.922, E3 -445477.005}
SPL {X  -159.990, Y  +562.598, Z    +0.000, E1  +337.958, E3 -445491.217}
SPL {X  -159.990, Y  +560.652, Z    +0.000, E1  +337.962, E3 -445501.429}
SPL {X  -159.990, Y  +558.143, Z    +0.000, E1  +337.928, E3 -445514.460}
SPL {X  -159.990, Y  +555.329, Z    +0.000, E1  +337.943, E3 -445529.205}
SPL {X  -159.990, Y  +553.115, Z    +0.000, E1  +337.946, E3 -445540.810}
SPL {X  -159.990, Y  +550.886, Z    +0.000, E1  +337.944, E3 -445552.491}
SPL {X  -159.990, Y  +548.568, Z    +0.000, E1  +337.944, E3 -445564.612}
SPL {X  -159.990, Y  +546.537, Z    +0.000, E1  +337.948, E3 -445575.247}
SPL {X  -159.990, Y  +545.062, Z    +0.000, E1  +337.955, E3 -445583.006}
SPL {X  -159.990, Y  +543.060, Z    +0.000, E1  +337.943, E3 -445593.485}
SPL {X  -159.990, Y  +539.928, Z    +0.000, E1  +337.917, E3 -445609.827}
SPL {X  -159.990, Y  +536.935, Z    +0.000, E1  +337.942, E3 -445625.544}
SPL {X  -159.990, Y  +534.656, Z    +0.000, E1  +337.946, E3 -445637.487}
SPL {X  -159.990, Y  +532.453, Z    +0.000, E1  +337.944, E3 -445649.014}
SPL {X  -159.990, Y  +530.660, Z    +0.000, E1  +337.952, E3 -445658.417}
SPL {X  -159.990, Y  +528.702, Z    +0.000, E1  +337.939, E3 -445668.630}
SPL {X  -159.990, Y  +525.760, Z    +0.000, E1  +337.914, E3 -445683.972}
SPL {X  -159.990, Y  +522.838, Z    +0.000, E1  +337.933, E3 -445699.338}
SPL {X  -159.990, Y  +520.708, Z    +0.000, E1  +337.953, E3 -445710.531}
SPL {X  -159.990, Y  +518.216, Z    +0.000, E1  +337.909, E3 -445723.449}
SPL {X  -159.990, Y  +515.568, Z    +0.000, E1  +338.084, E3 -445738.678}
ENDSPLINE

SPLINE
SPL {X  -159.990, Y  +518.374, Z    +0.000, E1  +341.240, E3 -445751.266}
ENDSPLINE

SPLINE
SPL {X  -159.990, Y  +513.606, Z    +0.000, E1  +339.879, E3 -445767.176}
SPL {X  -159.990, Y  +508.660, Z    +0.000, E1  +338.515, E3 -445782.606}
SPL {X  -159.990, Y  +505.237, Z    +0.000, E1  +337.606, E3 -445792.863}
SPL {X  -159.990, Y  +501.963, Z    +0.000, E1  +336.712, E3 -445801.967}
SPL {X  -159.990, Y  +498.406, Z    +0.000, E1  +335.789, E3 -445811.718}
SPL {X  -159.990, Y  +494.693, Z    +0.000, E1  +334.929, E3 -445822.185}
SPL {X  -159.990, Y  +491.649, Z    +0.000, E1  +334.596, E3 -445833.388}
SPL {X  -159.990, Y  +488.807, Z    +0.000, E1  +334.603, E3 -445846.112}
SPL {X  -159.990, Y  +486.070, Z    +0.000, E1  +334.601, E3 -445858.343}
SPL {X  -159.990, Y  +483.747, Z    +0.000, E1  +334.616, E3 -445868.756}
SPL {X  -159.990, Y  +481.980, Z    +0.000, E1  +334.616, E3 -445876.654}
SPL {X  -159.990, Y  +479.252, Z    +0.000, E1  +334.588, E3 -445888.795}
SPL {X  -159.990, Y  +475.940, Z    +0.000, E1  +334.597, E3 -445903.615}
SPL {X  -159.990, Y  +473.026, Z    +0.000, E1  +334.601, E3 -445916.645}
SPL {X  -159.990, Y  +470.047, Z    +0.000, E1  +334.598, E3 -445929.964}
SPL {X  -159.990, Y  +466.213, Z    +0.000, E1  +334.567, E3 -445947.043}
SPL {X  -159.990, Y  +462.520, Z    +0.000, E1  +334.600, E3 -445963.612}
SPL {X  -159.990, Y  +460.081, Z    +0.000, E1  +334.610, E3 -445974.513}
SPL {X  -159.990, Y  +457.497, Z    +0.000, E1  +334.597, E3 -445986.038}
SPL {X  -159.990, Y  +455.126, Z    +0.000, E1  +334.611, E3 -445996.646}
SPL {X  -159.990, Y  +452.123, Z    +0.000, E1  +334.574, E3 -446010.004}
SPL {X  -159.990, Y  +448.503, Z    +0.000, E1  +334.590, E3 -446026.205}
SPL {X  -159.990, Y  +445.882, Z    +0.000, E1  +334.615, E3 -446038.008}
SPL {X  -159.990, Y  +443.345, Z    +0.000, E1  +334.610, E3 -446049.390}
SPL {X  -159.990, Y  +441.077, Z    +0.000, E1  +334.631, E3 -446059.588}
SPL {X  -159.990, Y  +438.608, Z    +0.000, E1  +334.608, E3 -446070.585}
SPL {X  -159.990, Y  +434.852, Z    +0.000, E1  +334.585, E3 -446087.340}
SPL {X  -159.990, Y  +430.645, Z    +0.000, E1  +334.586, E3 -446106.159}
SPL {X  -159.990, Y  +426.865, Z    +0.000, E1  +334.602, E3 -446123.089}
SPL {X  -159.990, Y  +424.251, Z    +0.000, E1  +334.625, E3 -446134.826}
SPL {X  -159.990, Y  +421.010, Z    +0.000, E1  +334.582, E3 -446149.241}
SPL {X  -159.990, Y  +417.103, Z    +0.000, E1  +334.600, E3 -446166.744}
SPL {X  -159.990, Y  +413.684, Z    +0.000, E1  +334.603, E3 -446182.043}
SPL {X  -159.990, Y  +410.645, Z    +0.000, E1  +334.615, E3 -446195.655}
SPL {X  -159.990, Y  +407.450, Z    +0.000, E1  +334.599, E3 -446209.904}
SPL {X  -159.990, Y  +403.513, Z    +0.000, E1  +334.580, E3 -446227.457}
SPL {X  -159.990, Y  +400.403, Z    +0.000, E1  +334.620, E3 -446241.440}
SPL {X  -159.990, Y  +397.743, Z    +0.000, E1  +334.600, E3 -446253.309}
SPL {X  -159.990, Y  +394.848, Z    +0.000, E1  +334.621, E3 -446266.310}
SPL {X  -159.990, Y  +392.473, Z    +0.000, E1  +334.623, E3 -446276.937}
SPL {X  -159.990, Y  +390.187, Z    +0.000, E1  +334.622, E3 -446287.195}
SPL {X  -159.990, Y  +387.503, Z    +0.000, E1  +334.622, E3 -446299.190}
SPL {X  -159.990, Y  +384.711, Z    +0.000, E1  +334.612, E3 -446311.633}
SPL {X  -159.988, Y  +381.794, Z    +0.000, E1  +334.611, E3 -446324.668}
SPL {X  -159.958, Y  +379.279, Z    +0.000, E1  +334.625, E3 -446335.958}
SPL {X  -159.894, Y  +376.959, Z    +0.000, E1  +334.630, E3 -446346.403}
SPL {X  -159.765, Y  +374.027, Z    +0.000, E1  +334.633, E3 -446359.618}
SPL {X  -159.607, Y  +371.442, Z    +0.000, E1  +334.673, E3 -446371.393}
SPL {X  -159.379, Y  +368.534, Z    +0.000, E1  +334.684, E3 -446384.581}
SPL {X  -159.113, Y  +365.767, Z    +0.000, E1  +334.734, E3 -446397.221}
SPL {X  -158.798, Y  +363.007, Z    +0.000, E1  +334.761, E3 -446409.861}
SPL {X  -158.453, Y  +360.380, Z    +0.000, E1  +334.828, E3 -446422.005}
SPL {X  -158.127, Y  +358.155, Z    +0.000, E1  +334.874, E3 -446432.336}
SPL {X  -158.095, Y  +357.947, Z    +0.000, E1  +338.259, E3 -446463.908}
ENDSPLINE

